// TIA Portal V15.1 export
// export: Created 2024-06-21T08:41:00.046392Z, ExportSetting WithDefaults, DisplayName Totally Integrated Automation Portal, DisplayVersion V15.1 Update 5, DisplayName TIA Portal Openness, DisplayVersion V15.1 Update 5, DisplayName SINAMICS Startdrive Advanced, DisplayVersion V15.1, DisplayName G130, G150, S120, S150, SINAMICS MV, S210, DisplayVersion V15.1, DisplayName G110M, G120, G120C, G120D, G120P, DisplayVersion V15.1, DisplayName STEP 7 Professional, DisplayVersion V15.1 Update 5, DisplayName STEP 7 Safety, DisplayVersion V15.1, DisplayName WinCC Professional, DisplayVersion V15.1 Update 5, DisplayName SIMATIC Visualization Architect, DisplayVersion V15.1
FUNCTION_BLOCK "LPhoneAlarmReqString"   // FB2255, FBD
TITLE = LPhoneAlarmReq
{ S7_Optimized_Access := 'FALSE' }
AUTHOR : VCC
FAMILY : Function
VERSION : 0.1
// =============================================================================
// This Module Handles Phone Alarm Requests
// =============================================================================
// stored: AutoNumber false, IsIECCheckEnabled false, SetENOAutomatically False, UDAEnableTagReadback false
   VAR_INPUT
      I_PhoneAlarmReq1 { ExternalAccessible := 'False'; ExternalVisible := 'False'; ExternalWritable := 'False'} : Bool;   // Request Team Leader Andon From Loading Stn / Request PhoneAlarm For Station / Request PhoneAlarm
      I_PhoneAlarmReq2 { ExternalAccessible := 'False'; ExternalVisible := 'False'; ExternalWritable := 'False'} : Bool;   // Request Maintenance Andon From Loading Stn / Request PhoneAlarm For Station / Request PhoneAlarm
      I_PhoneAlarmReq3 { ExternalAccessible := 'False'; ExternalVisible := 'False'; ExternalWritable := 'False'} : Bool;   // Request PhoneAlarm For Station / Request PhoneAlarm
      I_PhoneAlarmReq4 { ExternalAccessible := 'False'; ExternalVisible := 'False'; ExternalWritable := 'False'} : Bool;   // Request PhoneAlarm For Station / Request PhoneAlarm
      I_PhoneAlarmReq5 { ExternalAccessible := 'False'; ExternalVisible := 'False'; ExternalWritable := 'False'} : Bool;   // Request PhoneAlarm For Station / Request PhoneAlarm
      I_PhoneAlarmReq6 { ExternalAccessible := 'False'; ExternalVisible := 'False'; ExternalWritable := 'False'} : Bool;   // Request PhoneAlarm For Station / Request PhoneAlarm
      I_PhoneAlarmReq7 { ExternalAccessible := 'False'; ExternalVisible := 'False'; ExternalWritable := 'False'} : Bool;   // Request PhoneAlarm For Station / Request PhoneAlarm
      I_PhoneAlarmReq8 { ExternalAccessible := 'False'; ExternalVisible := 'False'; ExternalWritable := 'False'} : Bool;   // Request PhoneAlarm For Station / Request PhoneAlarm
      I_PhoneAlarmReq9 { ExternalAccessible := 'False'; ExternalVisible := 'False'; ExternalWritable := 'False'} : Bool;   // Request PhoneAlarm For Station / Request PhoneAlarm
      I_PhoneAlarmReq10 { ExternalAccessible := 'False'; ExternalVisible := 'False'; ExternalWritable := 'False'} : Bool;   // Request PhoneAlarm For Station / Request PhoneAlarm
      I_PhoneAlarmReq11 { ExternalAccessible := 'False'; ExternalVisible := 'False'; ExternalWritable := 'False'} : Bool;   // Request PhoneAlarm For Station / Request PhoneAlarm
      I_PhoneAlarmReq12 { ExternalAccessible := 'False'; ExternalVisible := 'False'; ExternalWritable := 'False'} : Bool;   // Request PhoneAlarm For Station / Request PhoneAlarm
      I_PhoneAlarmReq13 { ExternalAccessible := 'False'; ExternalVisible := 'False'; ExternalWritable := 'False'} : Bool;   // Request PhoneAlarm For Station / Request PhoneAlarm
      I_PhoneAlarmReq14 { ExternalAccessible := 'False'; ExternalVisible := 'False'; ExternalWritable := 'False'} : Bool;   // Request PhoneAlarm For Station / Request PhoneAlarm
      I_PhoneAlarmReq15 { ExternalAccessible := 'False'; ExternalVisible := 'False'; ExternalWritable := 'False'} : Bool;   // Request PhoneAlarm For Station / Request PhoneAlarm
      I_PhoneAlarmReq16 { ExternalAccessible := 'False'; ExternalVisible := 'False'; ExternalWritable := 'False'} : Bool;   // Request PhoneAlarm For Station / Request PhoneAlarm
      C_MessageType1 { ExternalAccessible := 'False'; ExternalVisible := 'False'; ExternalWritable := 'False'} : String[20];   // Configuration Station / Configuration Message
      C_Message1 { ExternalAccessible := 'False'; ExternalVisible := 'False'; ExternalWritable := 'False'} : String[120];   // Configuration Station / Configuration Message
      C_MessageType2 { ExternalAccessible := 'False'; ExternalVisible := 'False'; ExternalWritable := 'False'} : String[20];   // Configuration Station / Configuration Message
      C_Message2 { ExternalAccessible := 'False'; ExternalVisible := 'False'; ExternalWritable := 'False'} : String[120];   // Configuration Station / Configuration Message
      C_MessageType3 { ExternalAccessible := 'False'; ExternalVisible := 'False'; ExternalWritable := 'False'} : String[20];   // Configuration Station / Configuration Message
      C_Message3 { ExternalAccessible := 'False'; ExternalVisible := 'False'; ExternalWritable := 'False'} : String[120];   // Configuration Station / Configuration Message
      C_MessageType4 { ExternalAccessible := 'False'; ExternalVisible := 'False'; ExternalWritable := 'False'} : String[20];   // Configuration Station / Configuration Message
      C_Message4 { ExternalAccessible := 'False'; ExternalVisible := 'False'; ExternalWritable := 'False'} : String[120];   // Configuration Station / Configuration Message
      C_MessageType5 { ExternalAccessible := 'False'; ExternalVisible := 'False'; ExternalWritable := 'False'} : String[20];   // Configuration Station / Configuration Message
      C_Message5 { ExternalAccessible := 'False'; ExternalVisible := 'False'; ExternalWritable := 'False'} : String[120];   // Configuration Station / Configuration Message
      C_MessageType6 { ExternalAccessible := 'False'; ExternalVisible := 'False'; ExternalWritable := 'False'} : String[20];   // Configuration Station / Configuration Message
      C_Message6 { ExternalAccessible := 'False'; ExternalVisible := 'False'; ExternalWritable := 'False'} : String[120];   // Configuration Station / Configuration Message
      C_MessageType7 { ExternalAccessible := 'False'; ExternalVisible := 'False'; ExternalWritable := 'False'} : String[20];   // Configuration Station / Configuration Message
      C_Message7 { ExternalAccessible := 'False'; ExternalVisible := 'False'; ExternalWritable := 'False'} : String[120];   // Configuration Station / Configuration Message
      C_MessageType8 { ExternalAccessible := 'False'; ExternalVisible := 'False'; ExternalWritable := 'False'} : String[20];   // Configuration Station / Configuration Message
      C_Message8 { ExternalAccessible := 'False'; ExternalVisible := 'False'; ExternalWritable := 'False'} : String[120];   // Configuration Station / Configuration Message
      C_MessageType9 { ExternalAccessible := 'False'; ExternalVisible := 'False'; ExternalWritable := 'False'} : String[20];   // Configuration Station / Configuration Message
      C_Message9 { ExternalAccessible := 'False'; ExternalVisible := 'False'; ExternalWritable := 'False'} : String[120];   // Configuration Station / Configuration Message
      C_MessageType10 { ExternalAccessible := 'False'; ExternalVisible := 'False'; ExternalWritable := 'False'} : String[20];   // Configuration Station / Configuration Message
      C_Message10 { ExternalAccessible := 'False'; ExternalVisible := 'False'; ExternalWritable := 'False'} : String[120];   // Configuration Station / Configuration Message
      C_MessageType11 { ExternalAccessible := 'False'; ExternalVisible := 'False'; ExternalWritable := 'False'} : String[20];   // Configuration Station / Configuration Message
      C_Message11 { ExternalAccessible := 'False'; ExternalVisible := 'False'; ExternalWritable := 'False'} : String[120];   // Configuration Station / Configuration Message
      C_MessageType12 { ExternalAccessible := 'False'; ExternalVisible := 'False'; ExternalWritable := 'False'} : String[20];   // Configuration Station / Configuration Message
      C_Message12 { ExternalAccessible := 'False'; ExternalVisible := 'False'; ExternalWritable := 'False'} : String[120];   // Configuration Station / Configuration Message
      C_MessageType13 { ExternalAccessible := 'False'; ExternalVisible := 'False'; ExternalWritable := 'False'} : String[20];   // Configuration Station / Configuration Message
      C_Message13 { ExternalAccessible := 'False'; ExternalVisible := 'False'; ExternalWritable := 'False'} : String[120];   // Configuration Station / Configuration Message
      C_MessageType14 { ExternalAccessible := 'False'; ExternalVisible := 'False'; ExternalWritable := 'False'} : String[20];   // Configuration Station / Configuration Message
      C_Message14 { ExternalAccessible := 'False'; ExternalVisible := 'False'; ExternalWritable := 'False'} : String[120];   // Configuration Station / Configuration Message
      C_MessageType15 { ExternalAccessible := 'False'; ExternalVisible := 'False'; ExternalWritable := 'False'} : String[20];   // Configuration Station / Configuration Message
      C_Message15 { ExternalAccessible := 'False'; ExternalVisible := 'False'; ExternalWritable := 'False'} : String[120];   // Configuration Station / Configuration Message
      C_MessageType16 { ExternalAccessible := 'False'; ExternalVisible := 'False'; ExternalWritable := 'False'} : String[20];   // Configuration Station / Configuration Message
      C_Message16 { ExternalAccessible := 'False'; ExternalVisible := 'False'; ExternalWritable := 'False'} : String[120];   // Configuration Station / Configuration Message
      C_VDCommRecvDB { ExternalAccessible := 'False'; ExternalVisible := 'False'; ExternalWritable := 'False'} : DB_ANY;   // VD communication system receive DB; Not to be used by application / VD communication system receive DB Not to be used by Application
      C_VDCommSendDB { ExternalAccessible := 'False'; ExternalVisible := 'False'; ExternalWritable := 'False'} : DB_ANY;   // VD communication system send DB; Not to be used by application / VD communication system send DB Not to be used by Application
      C_LocalRecvDB { ExternalAccessible := 'False'; ExternalVisible := 'False'; ExternalWritable := 'False'} : DB_ANY;   // Local DB To Store Received Data
      C_LocalSendDB { ExternalAccessible := 'False'; ExternalVisible := 'False'; ExternalWritable := 'False'} : DB_ANY;   // Local DB for send data; to be used by application / Local DB For Send Data Used By The Application
      C_SubSystem { ExternalAccessible := 'False'; ExternalVisible := 'False'; ExternalWritable := 'False'} : Int;   // Number to identify the subsystem / Identify Subsystem
      C_FilterMessage1 { ExternalAccessible := 'False'; ExternalVisible := 'False'; ExternalWritable := 'False'} : Time;   // Filter
      C_FilterMessage2 { ExternalAccessible := 'False'; ExternalVisible := 'False'; ExternalWritable := 'False'} : Time;   // Filter
      C_FilterMessage3 { ExternalAccessible := 'False'; ExternalVisible := 'False'; ExternalWritable := 'False'} : Time;   // Filter
      C_FilterMessage4 { ExternalAccessible := 'False'; ExternalVisible := 'False'; ExternalWritable := 'False'} : Time;   // Filter
      C_FilterMessage5 { ExternalAccessible := 'False'; ExternalVisible := 'False'; ExternalWritable := 'False'} : Time;   // Filter
      C_FilterMessage6 { ExternalAccessible := 'False'; ExternalVisible := 'False'; ExternalWritable := 'False'} : Time;   // Filter
      C_FilterMessage7 { ExternalAccessible := 'False'; ExternalVisible := 'False'; ExternalWritable := 'False'} : Time;   // Filter
      C_FilterMessage8 { ExternalAccessible := 'False'; ExternalVisible := 'False'; ExternalWritable := 'False'} : Time;   // Filter
      C_FilterMessage9 { ExternalAccessible := 'False'; ExternalVisible := 'False'; ExternalWritable := 'False'} : Time;   // Filter
      C_FilterMessage10 { ExternalAccessible := 'False'; ExternalVisible := 'False'; ExternalWritable := 'False'} : Time;   // Filter
      C_FilterMessage11 { ExternalAccessible := 'False'; ExternalVisible := 'False'; ExternalWritable := 'False'} : Time;   // Filter
      C_FilterMessage12 { ExternalAccessible := 'False'; ExternalVisible := 'False'; ExternalWritable := 'False'} : Time;   // Filter
      C_FilterMessage13 { ExternalAccessible := 'False'; ExternalVisible := 'False'; ExternalWritable := 'False'} : Time;   // Filter
      C_FilterMessage14 { ExternalAccessible := 'False'; ExternalVisible := 'False'; ExternalWritable := 'False'} : Time;   // Filter
      C_FilterMessage15 { ExternalAccessible := 'False'; ExternalVisible := 'False'; ExternalWritable := 'False'} : Time;   // Filter
      C_FilterMessage16 { ExternalAccessible := 'False'; ExternalVisible := 'False'; ExternalWritable := 'False'} : Time;   // Filter
   END_VAR
   VAR_IN_OUT
      IO_VD : "VDComm";   // Communication
      H_HMI : "H_HMI";   // Animation
      H_PhoneAlarmReqString : "H_PhoneAlarmReqString";   // Animation
   END_VAR
   VAR DB_SPECIFIC
      ReqPhoneAlarm { ExternalAccessible := 'False'; ExternalVisible := 'False'; ExternalWritable := 'False'} : Array[1..16] of Bool;   // Request Team Leader Andon / Request PhoneAlarm
      VDReqPhoneAlarm { ExternalAccessible := 'False'; ExternalVisible := 'False'; ExternalWritable := 'False'} : Array[1..16] of Bool;   // VD Request Team Leader Andon / VD Request PhoneAlarm
      Done { ExternalAccessible := 'False'; ExternalVisible := 'False'; ExternalWritable := 'False'} : Array[1..16] of Bool;   // Array
      StnEdge { ExternalAccessible := 'False'; ExternalVisible := 'False'; ExternalWritable := 'False'} : Array[1..16] of Bool;   // Pos Edge
      SendDoneToVD { ExternalAccessible := 'False'; ExternalVisible := 'False'; ExternalWritable := 'False'} : Bool;   // Request Is Finished
      SendVD { ExternalAccessible := 'False'; ExternalVisible := 'False'; ExternalWritable := 'False'} : Bool;   // Send
      PhoneAlarmReqActiveStn1 { ExternalAccessible := 'False'; ExternalVisible := 'False'; ExternalWritable := 'False'} : Bool;   // Indication Request Team Leader Andon / Indication Request
      PhoneAlarmReqActiveStn2 { ExternalAccessible := 'False'; ExternalVisible := 'False'; ExternalWritable := 'False'} : Bool;   // Indication Maintenance Andon / Indication Request
      PhoneAlarmReqActiveStn3 { ExternalAccessible := 'False'; ExternalVisible := 'False'; ExternalWritable := 'False'} : Bool;   // Indication Request
      PhoneAlarmReqActiveStn4 { ExternalAccessible := 'False'; ExternalVisible := 'False'; ExternalWritable := 'False'} : Bool;   // Indication Request
      PhoneAlarmReqActiveStn5 { ExternalAccessible := 'False'; ExternalVisible := 'False'; ExternalWritable := 'False'} : Bool;   // Indication Request
      PhoneAlarmReqActiveStn6 { ExternalAccessible := 'False'; ExternalVisible := 'False'; ExternalWritable := 'False'} : Bool;   // Indication Request
      PhoneAlarmReqActiveStn7 { ExternalAccessible := 'False'; ExternalVisible := 'False'; ExternalWritable := 'False'} : Bool;   // Indication Request
      PhoneAlarmReqActiveStn8 { ExternalAccessible := 'False'; ExternalVisible := 'False'; ExternalWritable := 'False'} : Bool;   // Indication Request
      PhoneAlarmReqActiveStn9 { ExternalAccessible := 'False'; ExternalVisible := 'False'; ExternalWritable := 'False'} : Bool;   // Indication Request
      PhoneAlarmReqActiveStn10 { ExternalAccessible := 'False'; ExternalVisible := 'False'; ExternalWritable := 'False'} : Bool;   // Indication Request
      PhoneAlarmReqActiveStn11 { ExternalAccessible := 'False'; ExternalVisible := 'False'; ExternalWritable := 'False'} : Bool;   // Indication Request
      PhoneAlarmReqActiveStn12 { ExternalAccessible := 'False'; ExternalVisible := 'False'; ExternalWritable := 'False'} : Bool;   // Indication Request
      PhoneAlarmReqActiveStn13 { ExternalAccessible := 'False'; ExternalVisible := 'False'; ExternalWritable := 'False'} : Bool;   // Indication Request
      PhoneAlarmReqActiveStn14 { ExternalAccessible := 'False'; ExternalVisible := 'False'; ExternalWritable := 'False'} : Bool;   // Indication Request
      PhoneAlarmReqActiveStn15 { ExternalAccessible := 'False'; ExternalVisible := 'False'; ExternalWritable := 'False'} : Bool;   // Indication Request
      PhoneAlarmReqActiveStn16 { ExternalAccessible := 'False'; ExternalVisible := 'False'; ExternalWritable := 'False'} : Bool;   // Indication Request
      VDMessage { ExternalAccessible := 'False'; ExternalVisible := 'False'; ExternalWritable := 'False'} : Struct   // VD MEssage to send
         VDMessageType { ExternalAccessible := 'False'; ExternalVisible := 'False'; ExternalWritable := 'False'} : Array[0..19] of Byte;   // Attention Event / VD MessageType
         VDMessage { ExternalAccessible := 'False'; ExternalVisible := 'False'; ExternalWritable := 'False'} : Array[0..119] of Byte;   // Attention Event / VD Message
      END_STRUCT;
   END_VAR
   VAR
      _VDComSubSystem { ExternalAccessible := 'False'; ExternalVisible := 'False'; ExternalWritable := 'False'; S7_SetPoint := 'True'} : "LVDComSubSystemS7-1500";   // FB
   END_VAR
   VAR DB_SPECIFIC
      Edge { ExternalAccessible := 'False'; ExternalVisible := 'False'; ExternalWritable := 'False'} : Array[0..15] of Bool;   // Array Edge
      InitDone { ExternalAccessible := 'False'; ExternalVisible := 'False'; ExternalWritable := 'False'} : Array[1..32] of Bool;   // Init Done
      InitDoneEdge { ExternalAccessible := 'False'; ExternalVisible := 'False'; ExternalWritable := 'False'} : Array[1..32] of Bool;   // Edge Done
      MessageType { ExternalAccessible := 'False'; ExternalVisible := 'False'; ExternalWritable := 'False'} : Int;   // Message Type
      MessageLength { ExternalAccessible := 'False'; ExternalVisible := 'False'; ExternalWritable := 'False'} : Word;   // Message Type / Message Lenght
      _Filter1 { ExternalAccessible := 'False'; ExternalVisible := 'False'; ExternalWritable := 'False'; S7_SetPoint := 'True'} : TON_TIME;   // FB
      _Filter2 { ExternalAccessible := 'False'; ExternalVisible := 'False'; ExternalWritable := 'False'; S7_SetPoint := 'True'} : TON_TIME;   // FB
      _Filter3 { ExternalAccessible := 'False'; ExternalVisible := 'False'; ExternalWritable := 'False'; S7_SetPoint := 'True'} : TON_TIME;   // FB
      _Filter4 { ExternalAccessible := 'False'; ExternalVisible := 'False'; ExternalWritable := 'False'; S7_SetPoint := 'True'} : TON_TIME;   // FB
      _Filter5 { ExternalAccessible := 'False'; ExternalVisible := 'False'; ExternalWritable := 'False'; S7_SetPoint := 'True'} : TON_TIME;   // FB
      _Filter6 { ExternalAccessible := 'False'; ExternalVisible := 'False'; ExternalWritable := 'False'; S7_SetPoint := 'True'} : TON_TIME;   // FB
      _Filter7 { ExternalAccessible := 'False'; ExternalVisible := 'False'; ExternalWritable := 'False'; S7_SetPoint := 'True'} : TON_TIME;   // FB
      _Filter8 { ExternalAccessible := 'False'; ExternalVisible := 'False'; ExternalWritable := 'False'; S7_SetPoint := 'True'} : TON_TIME;   // FB
      _Filter9 { ExternalAccessible := 'False'; ExternalVisible := 'False'; ExternalWritable := 'False'; S7_SetPoint := 'True'} : TON_TIME;   // FB
      _Filter10 { ExternalAccessible := 'False'; ExternalVisible := 'False'; ExternalWritable := 'False'; S7_SetPoint := 'True'} : TON_TIME;   // FB
      _Filter11 { ExternalAccessible := 'False'; ExternalVisible := 'False'; ExternalWritable := 'False'; S7_SetPoint := 'True'} : TON_TIME;   // FB
      _Filter12 { ExternalAccessible := 'False'; ExternalVisible := 'False'; ExternalWritable := 'False'; S7_SetPoint := 'True'} : TON_TIME;   // FB
      _Filter13 { ExternalAccessible := 'False'; ExternalVisible := 'False'; ExternalWritable := 'False'; S7_SetPoint := 'True'} : TON_TIME;   // FB
      _Filter14 { ExternalAccessible := 'False'; ExternalVisible := 'False'; ExternalWritable := 'False'; S7_SetPoint := 'True'} : TON_TIME;   // FB
      _Filter15 { ExternalAccessible := 'False'; ExternalVisible := 'False'; ExternalWritable := 'False'; S7_SetPoint := 'True'} : TON_TIME;   // FB
      _Filter16 { ExternalAccessible := 'False'; ExternalVisible := 'False'; ExternalWritable := 'False'; S7_SetPoint := 'True'} : TON_TIME;   // FB
      SendToVDTimeOut { ExternalAccessible := 'False'; ExternalVisible := 'False'; ExternalWritable := 'False'; S7_SetPoint := 'True'} : TON_TIME;   // Send to VD time-out
      ResetVDComm { ExternalAccessible := 'False'; ExternalVisible := 'False'; ExternalWritable := 'False'} : Bool;   // Reset VD communication upon timeout
      VDMessageTypeTemp { ExternalAccessible := 'False'; ExternalVisible := 'False'; ExternalWritable := 'False'} : String[20];   // Attention Event / VDMessageTypeTemp string 20 characters
      VDMessageTemp { ExternalAccessible := 'False'; ExternalVisible := 'False'; ExternalWritable := 'False'} : String[120];   // Attention Event / VDMessageTemp string 120 characters
      VDMessageTypeSerialzePos { ExternalAccessible := 'False'; ExternalVisible := 'False'; ExternalWritable := 'False'} : DInt;   // Serialize position
      VDMessageSerialzePos { ExternalAccessible := 'False'; ExternalVisible := 'False'; ExternalWritable := 'False'} : DInt;   // Serialize position
      VDMessageTypeTempArray { ExternalAccessible := 'False'; ExternalVisible := 'False'; ExternalWritable := 'False'} : Array[0..21] of Byte;   // VDMessageType Array
      VDMessageTempArray { ExternalAccessible := 'False'; ExternalVisible := 'False'; ExternalWritable := 'False'} : Array[0..121] of Byte;   // VDMessage Array
   END_VAR
   VAR_TEMP
      RequestCommand1 : Bool;   // Light On To Building Infrastructure / Request Configured Command
      RequestCommand2 : Bool;   // Light On To Building Infrastructure / Request Configured Command
      RequestCommand3 : Bool;   // Light On To Building Infrastructure / Request Configured Command
      RequestCommand4 : Bool;   // Light On To Building Infrastructure / Request Configured Command
      RequestCommand5 : Bool;   // Light On To Building Infrastructure / Request Configured Command
      RequestCommand6 : Bool;   // Light On To Building Infrastructure / Request Configured Command
      RequestCommand7 : Bool;   // Light On To Building Infrastructure / Request Configured Command
      RequestCommand8 : Bool;   // Light On To Building Infrastructure / Request Configured Command
      RequestCommand9 : Bool;   // Request Configured Command
      RequestCommand10 : Bool;   // Request Configured Command
      RequestCommand11 : Bool;   // Request Configured Command
      RequestCommand12 : Bool;   // Request Configured Command
      RequestCommand13 : Bool;   // Request Configured Command
      RequestCommand14 : Bool;   // Request Configured Command
      RequestCommand15 : Bool;   // Request Configured Command
      RequestCommand16 : Bool;   // Request Configured Command
      RecvDBNbr : Int;   // Receive system DB Number
      SendDBNbr : Int;   // Send system DB Number
      LocalRecvDBNbr : Int;   // Receive DB Number Local by Application
      LocalSendDBNbr : Int;   // Send DB Number Local by Application
      PtrASnd : Any;   // Pointer to the Application receive DB / Pointer to the Application send DB
   END_VAR
   VAR CONSTANT
      String20Spaces : String := '                    ';   // String with 20 spaces
      String120Spaces : String := '                                                                                                                        ';   // String with 120 spaces
   END_VAR
   VAR_TEMP   // added for the SCL form of the ladder/FBD networks
      _w1 : Bool;
      _w2 : Bool;
   END_VAR
BEGIN

REGION Network 1: **** 1 - Inputs **** Extract The Commands From HMI
   // Extract The Commands From HMI
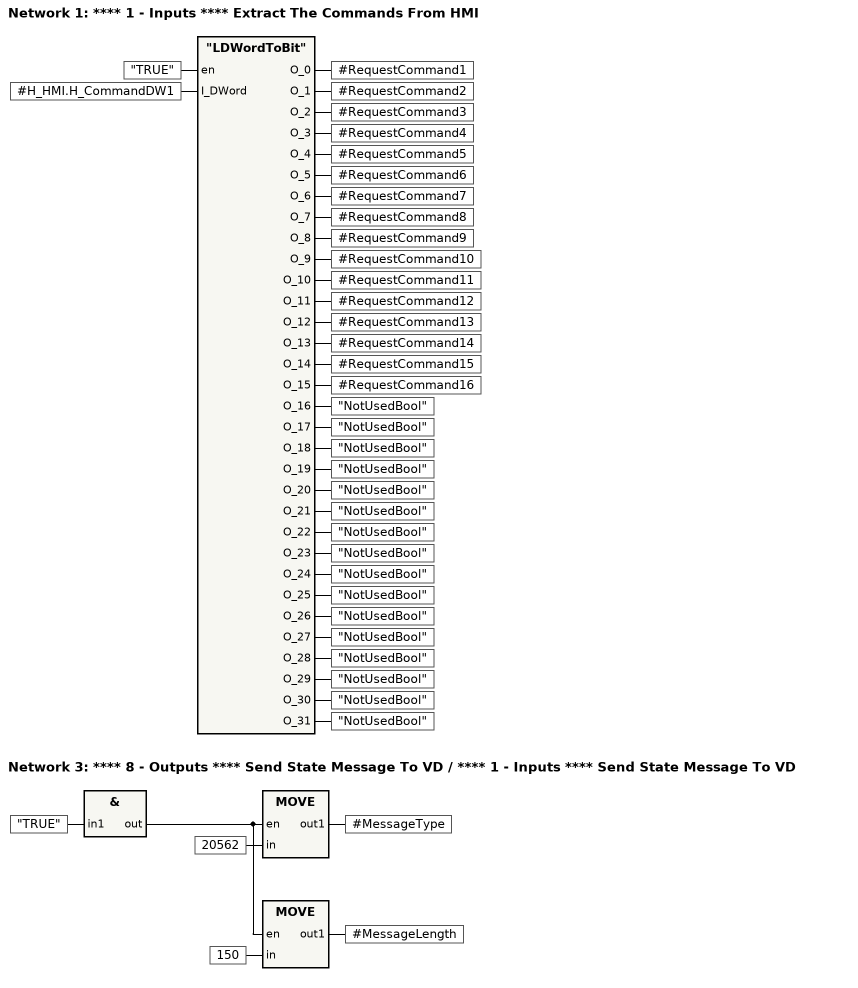
   IF "TRUE" THEN
       "LDWordToBit"(I_DWord := #H_HMI.H_CommandDW1,
                     O_0 => #RequestCommand1,
                     O_1 => #RequestCommand2,
                     O_2 => #RequestCommand3,
                     O_3 => #RequestCommand4,
                     O_4 => #RequestCommand5,
                     O_5 => #RequestCommand6,
                     O_6 => #RequestCommand7,
                     O_7 => #RequestCommand8,
                     O_8 => #RequestCommand9,
                     O_9 => #RequestCommand10,
                     O_10 => #RequestCommand11,
                     O_11 => #RequestCommand12,
                     O_12 => #RequestCommand13,
                     O_13 => #RequestCommand14,
                     O_14 => #RequestCommand15,
                     O_15 => #RequestCommand16,
                     O_16 => "NotUsedBool",
                     O_17 => "NotUsedBool",
                     O_18 => "NotUsedBool",
                     O_19 => "NotUsedBool",
                     O_20 => "NotUsedBool",
                     O_21 => "NotUsedBool",
                     O_22 => "NotUsedBool",
                     O_23 => "NotUsedBool",
                     O_24 => "NotUsedBool",
                     O_25 => "NotUsedBool",
                     O_26 => "NotUsedBool",
                     O_27 => "NotUsedBool",
                     O_28 => "NotUsedBool",
                     O_29 => "NotUsedBool",
                     O_30 => "NotUsedBool",
                     O_31 => "NotUsedBool");
   END_IF;
END_REGION

NETWORK
TITLE = **** 1 - Inputs **** Load DB / **** 1 - Inputs **** Load DB number
// Load DB numbers to local variables from the Receive and Send DB from - VD Master - VD Subsystem
// Read DB Number Recv
      OPN   #C_VDCommRecvDB;
      L     DBNO;
      T     #RecvDBNbr;

// Read DB Number Send
      OPN   #C_VDCommSendDB;
      L     DBNO;
      T     #SendDBNbr;

// DB Number from VD Sub system
      OPN   #C_LocalRecvDB;
      L     DBNO;
      T     #LocalRecvDBNbr;

// Read DB Number Send
      OPN   #C_LocalSendDB;
      L     DBNO;
      T     #LocalSendDBNbr;

REGION Network 3: **** 8 - Outputs **** Send State Message To VD / **** 1 - Inputs **** Send State Message To VD
   // Send State Message To VD
   IF "TRUE" THEN
       #MessageType := 20562;
       #MessageLength := 150;
   END_IF;
END_REGION

REGION Network 4: **** 3.1 - Communication - Other Systems **** Send Message
   // Send Message
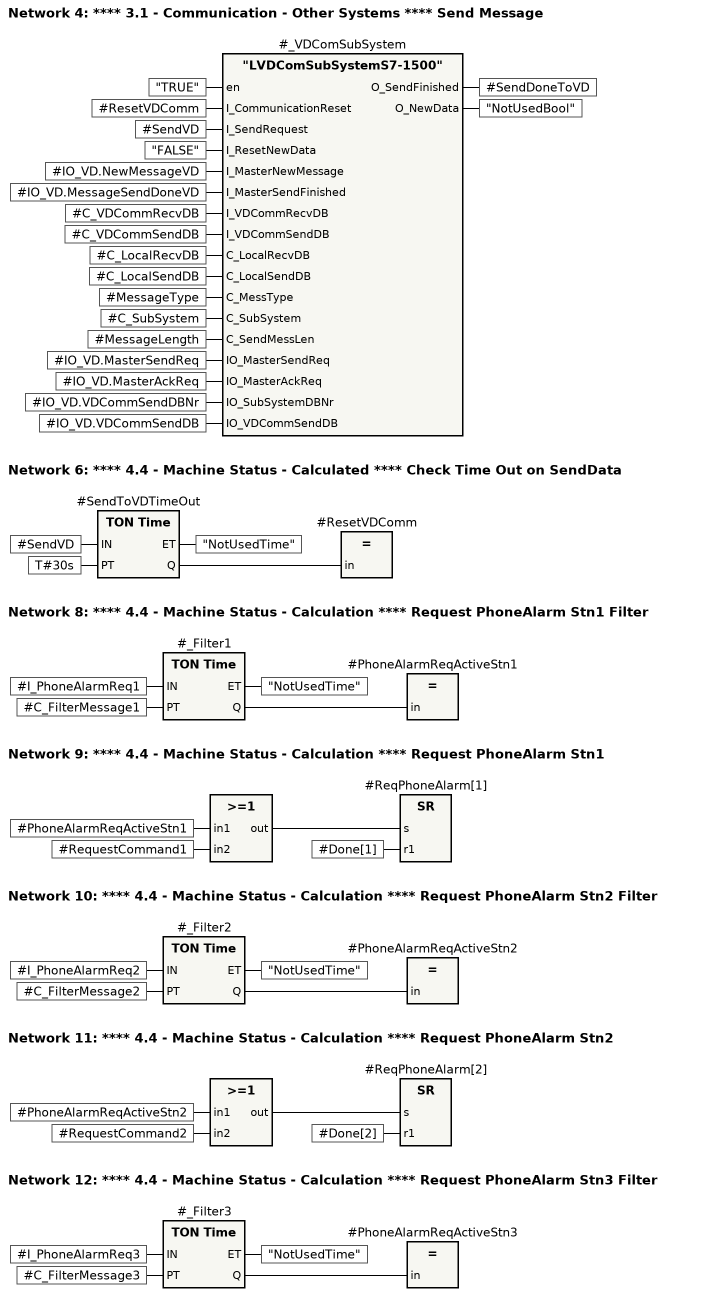
   IF "TRUE" THEN
       #_VDComSubSystem(I_CommunicationReset := #ResetVDComm,   // "LVDComSubSystemS7-1500"
                        I_SendRequest := #SendVD,
                        I_ResetNewData := "FALSE",
                        I_MasterNewMessage := #IO_VD.NewMessageVD,
                        I_MasterSendFinished := #IO_VD.MessageSendDoneVD,
                        I_VDCommRecvDB := #C_VDCommRecvDB,
                        I_VDCommSendDB := #C_VDCommSendDB,
                        C_LocalRecvDB := #C_LocalRecvDB,
                        C_LocalSendDB := #C_LocalSendDB,
                        C_MessType := #MessageType,
                        C_SubSystem := #C_SubSystem,
                        C_SendMessLen := #MessageLength,
                        IO_MasterSendReq := #IO_VD.MasterSendReq,
                        IO_MasterAckReq := #IO_VD.MasterAckReq,
                        IO_SubSystemDBNr := #IO_VD.VDCommSendDBNr,
                        IO_VDCommSendDB := #IO_VD.VDCommSendDB,
                        O_SendFinished => #SendDoneToVD,
                        O_NewData => "NotUsedBool");
   END_IF;
END_REGION

NETWORK
TITLE = **** 3.1 - Communication - Other Systems **** Configure DB / **** 4.2 Parameter **** Configure DB
// Configure DB pointers
      LAR1  P##PtrASnd;
      L     16#1002;  // Data type to copy B#16#2 = Bytes
      T     LW [AR1, P#0.0];
      L     #MessageLength;  //Length sending data
      T     LW [AR1, P#2.0];
      L     #LocalSendDBNbr;  // Local Send DB Number
      T     LW [AR1, P#4.0];
      L     10;  // Offset in DB (skip VD header)
      SLD   3;  // Convert to pointer - Shift Left DW
      OD    16#8400_0000;  // Memory area DB Memory - 84 equals DB
      T     LD [AR1, P#6.0];


REGION Network 6: **** 4.4 - Machine Status - Calculated **** Check Time Out on SendData
   // Reset Send request when time out elapses
   // Reset the VD communication
   #SendToVDTimeOut(IN := #SendVD, PT := T#30s, ET => "NotUsedTime");   // TON
   #ResetVDComm := #SendToVDTimeOut.Q;
END_REGION

NETWORK
TITLE = **** 4.4 - Machine status - Calculated **** Init Done
// Init Done

      A     #I_PhoneAlarmReq1;
      O     #RequestCommand1;
      FP    #InitDoneEdge[1];
      =     #InitDone[1];

      A     #I_PhoneAlarmReq2;
      O     #RequestCommand2;
      FP    #InitDoneEdge[2];
      =     #InitDone[2];

      A     #I_PhoneAlarmReq3;
      O     #RequestCommand3;
      FP    #InitDoneEdge[3];
      =     #InitDone[3];

      A     #I_PhoneAlarmReq4;
      O     #RequestCommand4;
      FP    #InitDoneEdge[4];
      =     #InitDone[4];

      A     #I_PhoneAlarmReq5;
      O     #RequestCommand5;
      FP    #InitDoneEdge[5];
      =     #InitDone[5];

      A     #I_PhoneAlarmReq6;
      O     #RequestCommand6;
      FP    #InitDoneEdge[6];
      =     #InitDone[6];

      A     #I_PhoneAlarmReq7;
      O     #RequestCommand7;
      FP    #InitDoneEdge[7];
      =     #InitDone[7];

      A     #I_PhoneAlarmReq8;
      O     #RequestCommand8;
      FP    #InitDoneEdge[8];
      =     #InitDone[8];

      A     #I_PhoneAlarmReq9;
      O     #RequestCommand9;
      FP    #InitDoneEdge[9];
      =     #InitDone[9];

      A     #I_PhoneAlarmReq10;
      O     #RequestCommand10;
      FP    #InitDoneEdge[10];
      =     #InitDone[10];

      A     #I_PhoneAlarmReq11;
      O     #RequestCommand11;
      FP    #InitDoneEdge[11];
      =     #InitDone[11];

      A     #I_PhoneAlarmReq12;
      O     #RequestCommand12;
      FP    #InitDoneEdge[12];
      =     #InitDone[12];

      A     #I_PhoneAlarmReq13;
      O     #RequestCommand13;
      FP    #InitDoneEdge[13];
      =     #InitDone[13];

      A     #I_PhoneAlarmReq14;
      O     #RequestCommand14;
      FP    #InitDoneEdge[14];
      =     #InitDone[14];

      A     #I_PhoneAlarmReq15;
      O     #RequestCommand15;
      FP    #InitDoneEdge[15];
      =     #InitDone[15];

      A     #I_PhoneAlarmReq16;
      O     #RequestCommand16;
      FP    #InitDoneEdge[16];
      =     #InitDone[16];


REGION Network 8: **** 4.4 - Machine Status - Calculation **** Request PhoneAlarm Stn1 Filter
   // Filter
   #_Filter1(IN := #I_PhoneAlarmReq1, PT := #C_FilterMessage1, ET => "NotUsedTime");   // TON
   #PhoneAlarmReqActiveStn1 := #_Filter1.Q;
END_REGION

REGION Network 9: **** 4.4 - Machine Status - Calculation **** Request PhoneAlarm Stn1
   // Request PhoneAlarm Stn1
   IF #PhoneAlarmReqActiveStn1 OR #RequestCommand1 THEN
       #ReqPhoneAlarm[1] := TRUE;   // SR flip-flop
   END_IF;
   IF #Done[1] THEN #ReqPhoneAlarm[1] := FALSE; END_IF;
END_REGION

REGION Network 10: **** 4.4 - Machine Status - Calculation **** Request PhoneAlarm Stn2 Filter
   // Filter
   #_Filter2(IN := #I_PhoneAlarmReq2, PT := #C_FilterMessage2, ET => "NotUsedTime");   // TON
   #PhoneAlarmReqActiveStn2 := #_Filter2.Q;
END_REGION

REGION Network 11: **** 4.4 - Machine Status - Calculation **** Request PhoneAlarm Stn2
   // Request PhoneAlarm Stn2
   IF #PhoneAlarmReqActiveStn2 OR #RequestCommand2 THEN
       #ReqPhoneAlarm[2] := TRUE;   // SR flip-flop
   END_IF;
   IF #Done[2] THEN #ReqPhoneAlarm[2] := FALSE; END_IF;
END_REGION

REGION Network 12: **** 4.4 - Machine Status - Calculation **** Request PhoneAlarm Stn3 Filter
   // Filter
   #_Filter3(IN := #I_PhoneAlarmReq3, PT := #C_FilterMessage3, ET => "NotUsedTime");   // TON
   #PhoneAlarmReqActiveStn3 := #_Filter3.Q;
END_REGION

REGION Network 13: **** 4.4 - Machine Status - Calculation **** Request PhoneAlarm Stn3
   // Request PhoneAlarm Stn3
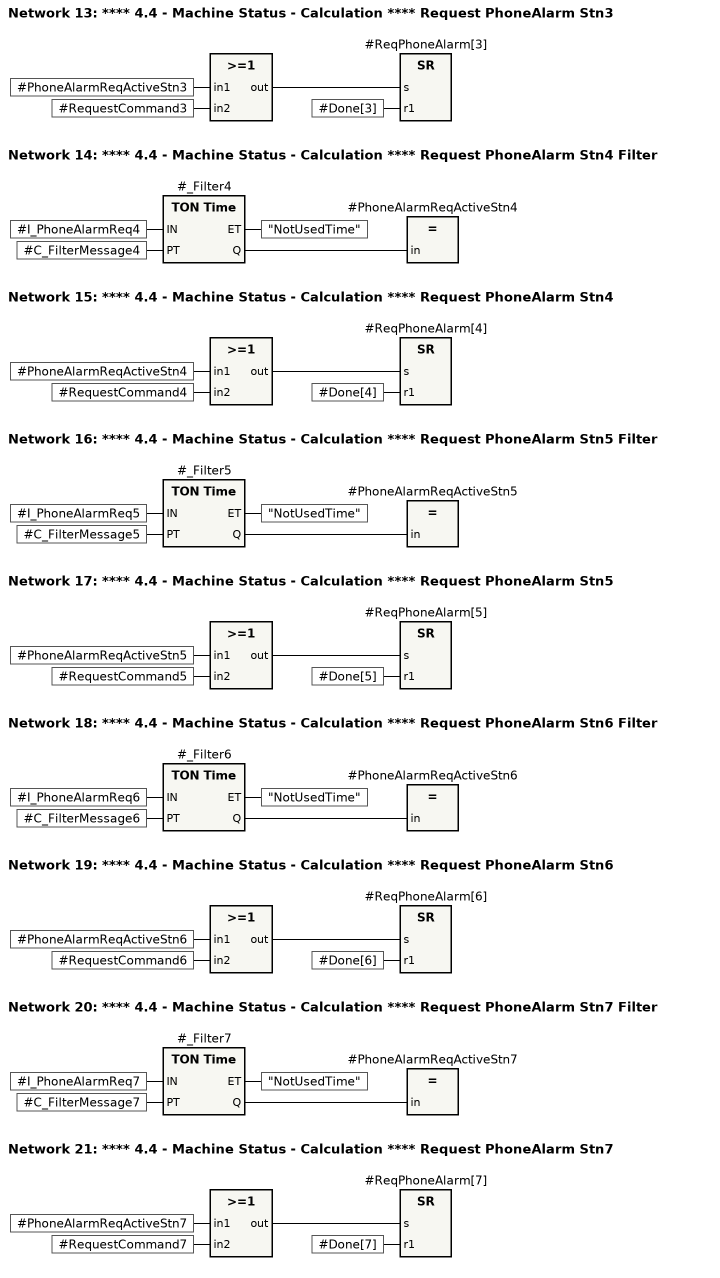
   IF #PhoneAlarmReqActiveStn3 OR #RequestCommand3 THEN
       #ReqPhoneAlarm[3] := TRUE;   // SR flip-flop
   END_IF;
   IF #Done[3] THEN #ReqPhoneAlarm[3] := FALSE; END_IF;
END_REGION

REGION Network 14: **** 4.4 - Machine Status - Calculation **** Request PhoneAlarm Stn4 Filter
   // Filter
   #_Filter4(IN := #I_PhoneAlarmReq4, PT := #C_FilterMessage4, ET => "NotUsedTime");   // TON
   #PhoneAlarmReqActiveStn4 := #_Filter4.Q;
END_REGION

REGION Network 15: **** 4.4 - Machine Status - Calculation **** Request PhoneAlarm Stn4
   // Request PhoneAlarm Stn4
   IF #PhoneAlarmReqActiveStn4 OR #RequestCommand4 THEN
       #ReqPhoneAlarm[4] := TRUE;   // SR flip-flop
   END_IF;
   IF #Done[4] THEN #ReqPhoneAlarm[4] := FALSE; END_IF;
END_REGION

REGION Network 16: **** 4.4 - Machine Status - Calculation **** Request PhoneAlarm Stn5 Filter
   // Filter
   #_Filter5(IN := #I_PhoneAlarmReq5, PT := #C_FilterMessage5, ET => "NotUsedTime");   // TON
   #PhoneAlarmReqActiveStn5 := #_Filter5.Q;
END_REGION

REGION Network 17: **** 4.4 - Machine Status - Calculation **** Request PhoneAlarm Stn5
   // Request PhoneAlarm Stn5
   IF #PhoneAlarmReqActiveStn5 OR #RequestCommand5 THEN
       #ReqPhoneAlarm[5] := TRUE;   // SR flip-flop
   END_IF;
   IF #Done[5] THEN #ReqPhoneAlarm[5] := FALSE; END_IF;
END_REGION

REGION Network 18: **** 4.4 - Machine Status - Calculation **** Request PhoneAlarm Stn6 Filter
   // Filter
   #_Filter6(IN := #I_PhoneAlarmReq6, PT := #C_FilterMessage6, ET => "NotUsedTime");   // TON
   #PhoneAlarmReqActiveStn6 := #_Filter6.Q;
END_REGION

REGION Network 19: **** 4.4 - Machine Status - Calculation **** Request PhoneAlarm Stn6
   // Request PhoneAlarm Stn6
   IF #PhoneAlarmReqActiveStn6 OR #RequestCommand6 THEN
       #ReqPhoneAlarm[6] := TRUE;   // SR flip-flop
   END_IF;
   IF #Done[6] THEN #ReqPhoneAlarm[6] := FALSE; END_IF;
END_REGION

REGION Network 20: **** 4.4 - Machine Status - Calculation **** Request PhoneAlarm Stn7 Filter
   // Filter
   #_Filter7(IN := #I_PhoneAlarmReq7, PT := #C_FilterMessage7, ET => "NotUsedTime");   // TON
   #PhoneAlarmReqActiveStn7 := #_Filter7.Q;
END_REGION

REGION Network 21: **** 4.4 - Machine Status - Calculation **** Request PhoneAlarm Stn7
   // Request PhoneAlarm Stn7
   IF #PhoneAlarmReqActiveStn7 OR #RequestCommand7 THEN
       #ReqPhoneAlarm[7] := TRUE;   // SR flip-flop
   END_IF;
   IF #Done[7] THEN #ReqPhoneAlarm[7] := FALSE; END_IF;
END_REGION

REGION Network 22: **** 4.4 - Machine Status - Calculation **** Request PhoneAlarm Stn8 Filter
   // Filter
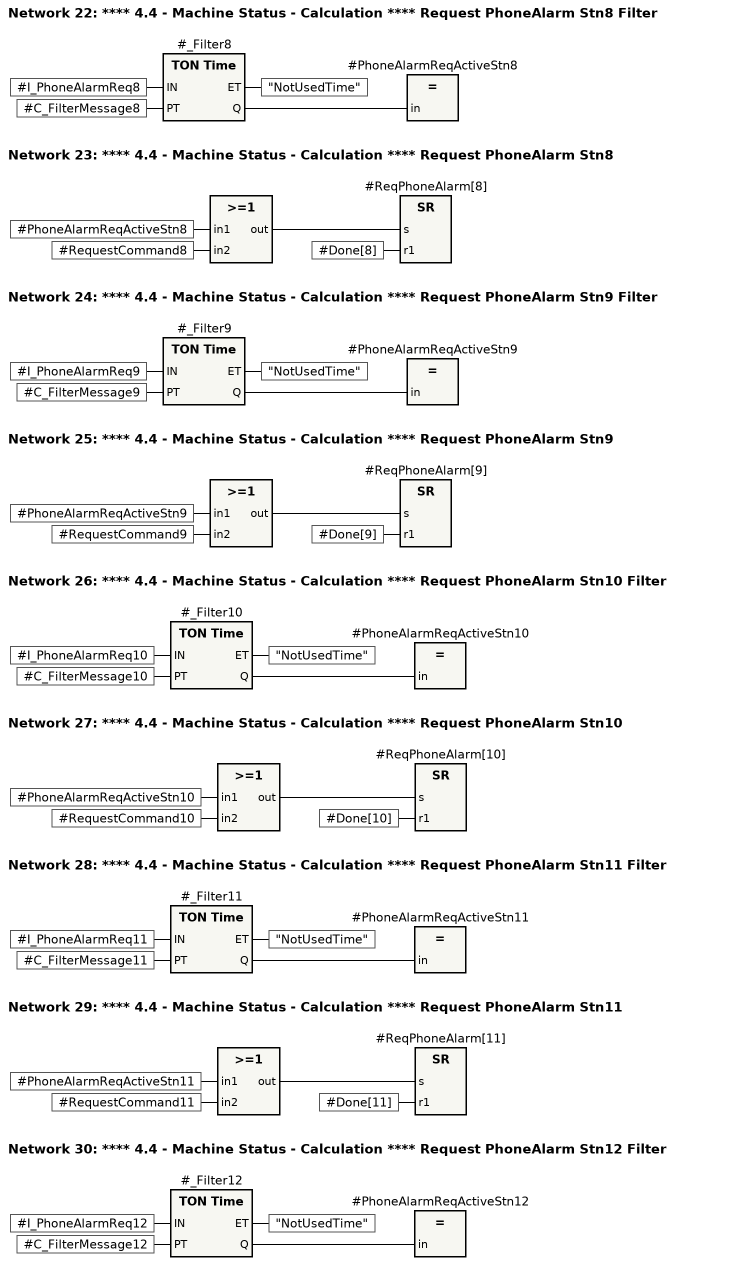
   #_Filter8(IN := #I_PhoneAlarmReq8, PT := #C_FilterMessage8, ET => "NotUsedTime");   // TON
   #PhoneAlarmReqActiveStn8 := #_Filter8.Q;
END_REGION

REGION Network 23: **** 4.4 - Machine Status - Calculation **** Request PhoneAlarm Stn8
   // Request PhoneAlarm Stn8
   IF #PhoneAlarmReqActiveStn8 OR #RequestCommand8 THEN
       #ReqPhoneAlarm[8] := TRUE;   // SR flip-flop
   END_IF;
   IF #Done[8] THEN #ReqPhoneAlarm[8] := FALSE; END_IF;
END_REGION

REGION Network 24: **** 4.4 - Machine Status - Calculation **** Request PhoneAlarm Stn9 Filter
   // Filter
   #_Filter9(IN := #I_PhoneAlarmReq9, PT := #C_FilterMessage9, ET => "NotUsedTime");   // TON
   #PhoneAlarmReqActiveStn9 := #_Filter9.Q;
END_REGION

REGION Network 25: **** 4.4 - Machine Status - Calculation **** Request PhoneAlarm Stn9
   // Request PhoneAlarm Stn9
   IF #PhoneAlarmReqActiveStn9 OR #RequestCommand9 THEN
       #ReqPhoneAlarm[9] := TRUE;   // SR flip-flop
   END_IF;
   IF #Done[9] THEN #ReqPhoneAlarm[9] := FALSE; END_IF;
END_REGION

REGION Network 26: **** 4.4 - Machine Status - Calculation **** Request PhoneAlarm Stn10 Filter
   // Filter
   #_Filter10(IN := #I_PhoneAlarmReq10, PT := #C_FilterMessage10, ET => "NotUsedTime");   // TON
   #PhoneAlarmReqActiveStn10 := #_Filter10.Q;
END_REGION

REGION Network 27: **** 4.4 - Machine Status - Calculation **** Request PhoneAlarm Stn10
   // Request PhoneAlarm Stn10
   IF #PhoneAlarmReqActiveStn10 OR #RequestCommand10 THEN
       #ReqPhoneAlarm[10] := TRUE;   // SR flip-flop
   END_IF;
   IF #Done[10] THEN #ReqPhoneAlarm[10] := FALSE; END_IF;
END_REGION

REGION Network 28: **** 4.4 - Machine Status - Calculation **** Request PhoneAlarm Stn11 Filter
   // Filter
   #_Filter11(IN := #I_PhoneAlarmReq11, PT := #C_FilterMessage11, ET => "NotUsedTime");   // TON
   #PhoneAlarmReqActiveStn11 := #_Filter11.Q;
END_REGION

REGION Network 29: **** 4.4 - Machine Status - Calculation **** Request PhoneAlarm Stn11
   // Request PhoneAlarm Stn11
   IF #PhoneAlarmReqActiveStn11 OR #RequestCommand11 THEN
       #ReqPhoneAlarm[11] := TRUE;   // SR flip-flop
   END_IF;
   IF #Done[11] THEN #ReqPhoneAlarm[11] := FALSE; END_IF;
END_REGION

REGION Network 30: **** 4.4 - Machine Status - Calculation **** Request PhoneAlarm Stn12 Filter
   // Filter
   #_Filter12(IN := #I_PhoneAlarmReq12, PT := #C_FilterMessage12, ET => "NotUsedTime");   // TON
   #PhoneAlarmReqActiveStn12 := #_Filter12.Q;
END_REGION

REGION Network 31: **** 4.4 - Machine Status - Calculation **** Request PhoneAlarm Stn12
   // Request PhoneAlarm Stn12
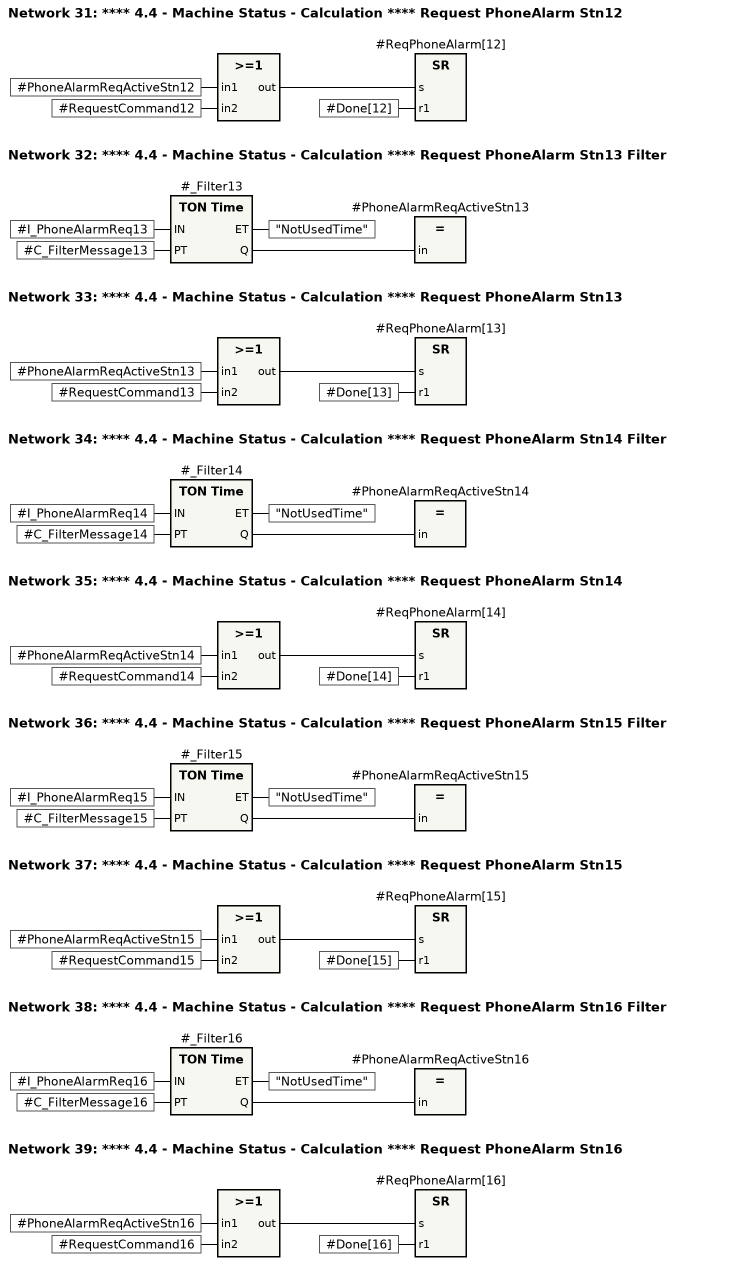
   IF #PhoneAlarmReqActiveStn12 OR #RequestCommand12 THEN
       #ReqPhoneAlarm[12] := TRUE;   // SR flip-flop
   END_IF;
   IF #Done[12] THEN #ReqPhoneAlarm[12] := FALSE; END_IF;
END_REGION

REGION Network 32: **** 4.4 - Machine Status - Calculation **** Request PhoneAlarm Stn13 Filter
   // Filter
   #_Filter13(IN := #I_PhoneAlarmReq13, PT := #C_FilterMessage13, ET => "NotUsedTime");   // TON
   #PhoneAlarmReqActiveStn13 := #_Filter13.Q;
END_REGION

REGION Network 33: **** 4.4 - Machine Status - Calculation **** Request PhoneAlarm Stn13
   // Request PhoneAlarm Stn13
   IF #PhoneAlarmReqActiveStn13 OR #RequestCommand13 THEN
       #ReqPhoneAlarm[13] := TRUE;   // SR flip-flop
   END_IF;
   IF #Done[13] THEN #ReqPhoneAlarm[13] := FALSE; END_IF;
END_REGION

REGION Network 34: **** 4.4 - Machine Status - Calculation **** Request PhoneAlarm Stn14 Filter
   // Filter
   #_Filter14(IN := #I_PhoneAlarmReq14, PT := #C_FilterMessage14, ET => "NotUsedTime");   // TON
   #PhoneAlarmReqActiveStn14 := #_Filter14.Q;
END_REGION

REGION Network 35: **** 4.4 - Machine Status - Calculation **** Request PhoneAlarm Stn14
   // Request PhoneAlarm Stn14
   IF #PhoneAlarmReqActiveStn14 OR #RequestCommand14 THEN
       #ReqPhoneAlarm[14] := TRUE;   // SR flip-flop
   END_IF;
   IF #Done[14] THEN #ReqPhoneAlarm[14] := FALSE; END_IF;
END_REGION

REGION Network 36: **** 4.4 - Machine Status - Calculation **** Request PhoneAlarm Stn15 Filter
   // Filter
   #_Filter15(IN := #I_PhoneAlarmReq15, PT := #C_FilterMessage15, ET => "NotUsedTime");   // TON
   #PhoneAlarmReqActiveStn15 := #_Filter15.Q;
END_REGION

REGION Network 37: **** 4.4 - Machine Status - Calculation **** Request PhoneAlarm Stn15
   // Request PhoneAlarm Stn15
   IF #PhoneAlarmReqActiveStn15 OR #RequestCommand15 THEN
       #ReqPhoneAlarm[15] := TRUE;   // SR flip-flop
   END_IF;
   IF #Done[15] THEN #ReqPhoneAlarm[15] := FALSE; END_IF;
END_REGION

REGION Network 38: **** 4.4 - Machine Status - Calculation **** Request PhoneAlarm Stn16 Filter
   // Filter
   #_Filter16(IN := #I_PhoneAlarmReq16, PT := #C_FilterMessage16, ET => "NotUsedTime");   // TON
   #PhoneAlarmReqActiveStn16 := #_Filter16.Q;
END_REGION

REGION Network 39: **** 4.4 - Machine Status - Calculation **** Request PhoneAlarm Stn16
   // Request PhoneAlarm Stn16
   IF #PhoneAlarmReqActiveStn16 OR #RequestCommand16 THEN
       #ReqPhoneAlarm[16] := TRUE;   // SR flip-flop
   END_IF;
   IF #Done[16] THEN #ReqPhoneAlarm[16] := FALSE; END_IF;
END_REGION

REGION Network 40: **** 4.4 - Machine Status - Calculation **** Message Request Done
   // Message Request Done
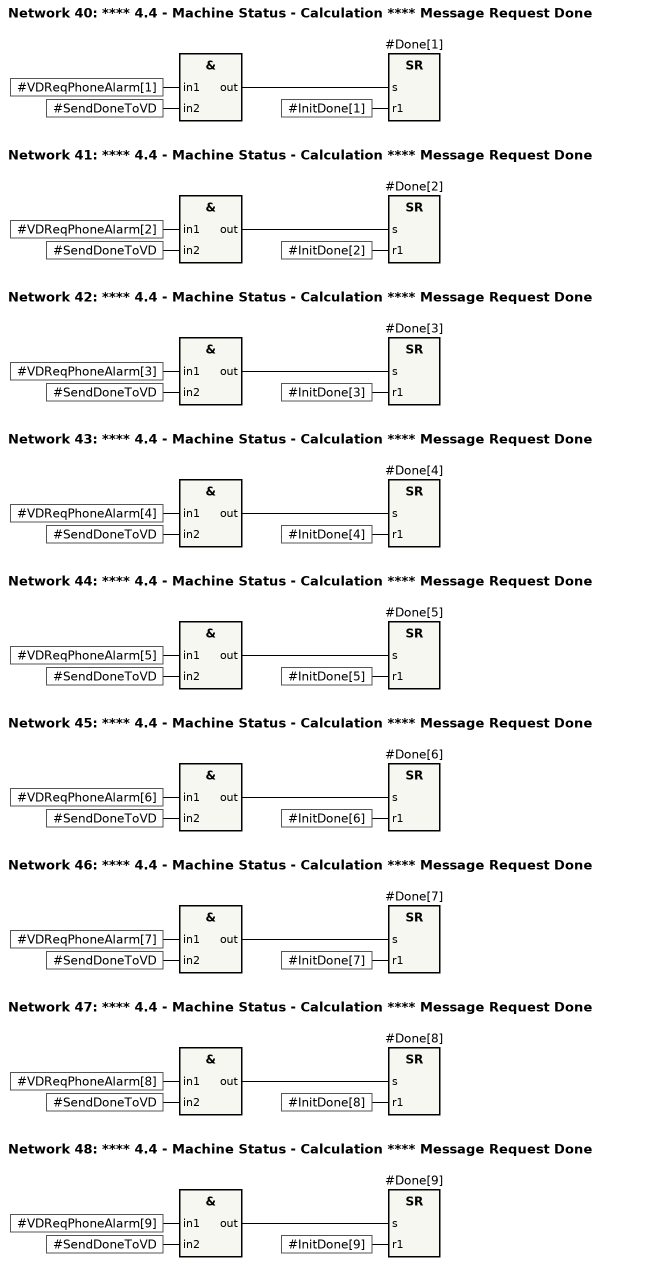
   IF #VDReqPhoneAlarm[1] AND #SendDoneToVD THEN
       #Done[1] := TRUE;   // SR flip-flop
   END_IF;
   IF #InitDone[1] THEN #Done[1] := FALSE; END_IF;
END_REGION

REGION Network 41: **** 4.4 - Machine Status - Calculation **** Message Request Done
   // Message Request Done
   IF #VDReqPhoneAlarm[2] AND #SendDoneToVD THEN
       #Done[2] := TRUE;   // SR flip-flop
   END_IF;
   IF #InitDone[2] THEN #Done[2] := FALSE; END_IF;
END_REGION

REGION Network 42: **** 4.4 - Machine Status - Calculation **** Message Request Done
   // Message Request Done
   IF #VDReqPhoneAlarm[3] AND #SendDoneToVD THEN
       #Done[3] := TRUE;   // SR flip-flop
   END_IF;
   IF #InitDone[3] THEN #Done[3] := FALSE; END_IF;
END_REGION

REGION Network 43: **** 4.4 - Machine Status - Calculation **** Message Request Done
   // Message Request Done
   IF #VDReqPhoneAlarm[4] AND #SendDoneToVD THEN
       #Done[4] := TRUE;   // SR flip-flop
   END_IF;
   IF #InitDone[4] THEN #Done[4] := FALSE; END_IF;
END_REGION

REGION Network 44: **** 4.4 - Machine Status - Calculation **** Message Request Done
   // Message Request Done
   IF #VDReqPhoneAlarm[5] AND #SendDoneToVD THEN
       #Done[5] := TRUE;   // SR flip-flop
   END_IF;
   IF #InitDone[5] THEN #Done[5] := FALSE; END_IF;
END_REGION

REGION Network 45: **** 4.4 - Machine Status - Calculation **** Message Request Done
   // Message Request Done
   IF #VDReqPhoneAlarm[6] AND #SendDoneToVD THEN
       #Done[6] := TRUE;   // SR flip-flop
   END_IF;
   IF #InitDone[6] THEN #Done[6] := FALSE; END_IF;
END_REGION

REGION Network 46: **** 4.4 - Machine Status - Calculation **** Message Request Done
   // Message Request Done
   IF #VDReqPhoneAlarm[7] AND #SendDoneToVD THEN
       #Done[7] := TRUE;   // SR flip-flop
   END_IF;
   IF #InitDone[7] THEN #Done[7] := FALSE; END_IF;
END_REGION

REGION Network 47: **** 4.4 - Machine Status - Calculation **** Message Request Done
   // Message Request Done
   IF #VDReqPhoneAlarm[8] AND #SendDoneToVD THEN
       #Done[8] := TRUE;   // SR flip-flop
   END_IF;
   IF #InitDone[8] THEN #Done[8] := FALSE; END_IF;
END_REGION

REGION Network 48: **** 4.4 - Machine Status - Calculation **** Message Request Done
   // Message Request Done
   IF #VDReqPhoneAlarm[9] AND #SendDoneToVD THEN
       #Done[9] := TRUE;   // SR flip-flop
   END_IF;
   IF #InitDone[9] THEN #Done[9] := FALSE; END_IF;
END_REGION

REGION Network 49: **** 4.4 - Machine Status - Calculation **** Message Request Done
   // Message Request Done
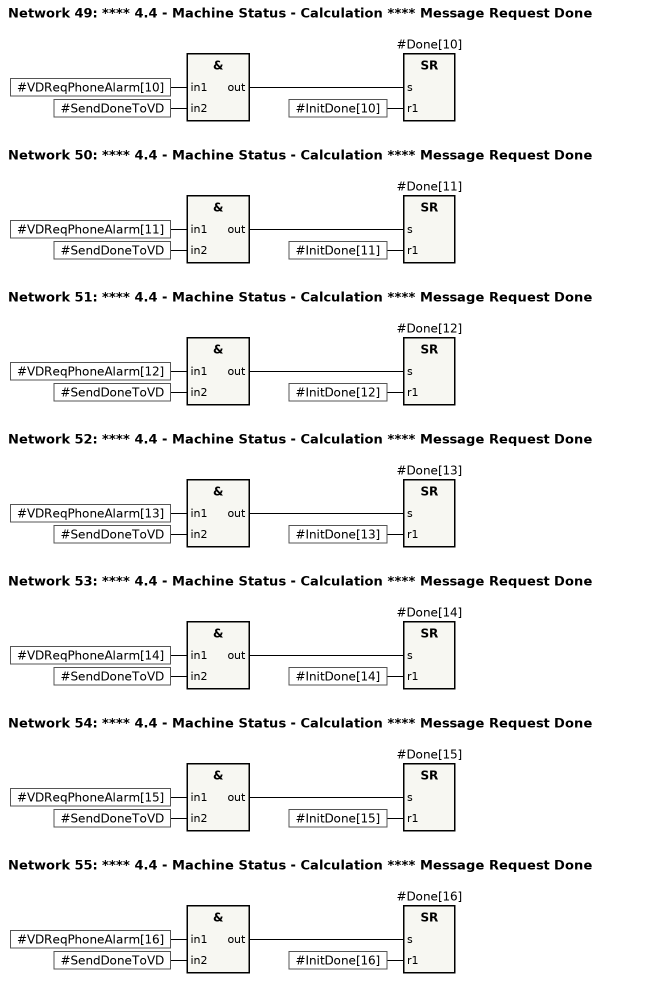
   IF #VDReqPhoneAlarm[10] AND #SendDoneToVD THEN
       #Done[10] := TRUE;   // SR flip-flop
   END_IF;
   IF #InitDone[10] THEN #Done[10] := FALSE; END_IF;
END_REGION

REGION Network 50: **** 4.4 - Machine Status - Calculation **** Message Request Done
   // Message Request Done
   IF #VDReqPhoneAlarm[11] AND #SendDoneToVD THEN
       #Done[11] := TRUE;   // SR flip-flop
   END_IF;
   IF #InitDone[11] THEN #Done[11] := FALSE; END_IF;
END_REGION

REGION Network 51: **** 4.4 - Machine Status - Calculation **** Message Request Done
   // Message Request Done
   IF #VDReqPhoneAlarm[12] AND #SendDoneToVD THEN
       #Done[12] := TRUE;   // SR flip-flop
   END_IF;
   IF #InitDone[12] THEN #Done[12] := FALSE; END_IF;
END_REGION

REGION Network 52: **** 4.4 - Machine Status - Calculation **** Message Request Done
   // Message Request Done
   IF #VDReqPhoneAlarm[13] AND #SendDoneToVD THEN
       #Done[13] := TRUE;   // SR flip-flop
   END_IF;
   IF #InitDone[13] THEN #Done[13] := FALSE; END_IF;
END_REGION

REGION Network 53: **** 4.4 - Machine Status - Calculation **** Message Request Done
   // Message Request Done
   IF #VDReqPhoneAlarm[14] AND #SendDoneToVD THEN
       #Done[14] := TRUE;   // SR flip-flop
   END_IF;
   IF #InitDone[14] THEN #Done[14] := FALSE; END_IF;
END_REGION

REGION Network 54: **** 4.4 - Machine Status - Calculation **** Message Request Done
   // Message Request Done
   IF #VDReqPhoneAlarm[15] AND #SendDoneToVD THEN
       #Done[15] := TRUE;   // SR flip-flop
   END_IF;
   IF #InitDone[15] THEN #Done[15] := FALSE; END_IF;
END_REGION

REGION Network 55: **** 4.4 - Machine Status - Calculation **** Message Request Done
   // Message Request Done
   IF #VDReqPhoneAlarm[16] AND #SendDoneToVD THEN
       #Done[16] := TRUE;   // SR flip-flop
   END_IF;
   IF #InitDone[16] THEN #Done[16] := FALSE; END_IF;
END_REGION

REGION Network 56: **** 4.4 - Machine Status - Calculation **** Que Message Request 1 / **** 4.4 - Machine Status - Calculation **** Queue Message Request 1
   // Que Message Request 1 / Queue Message Request 1
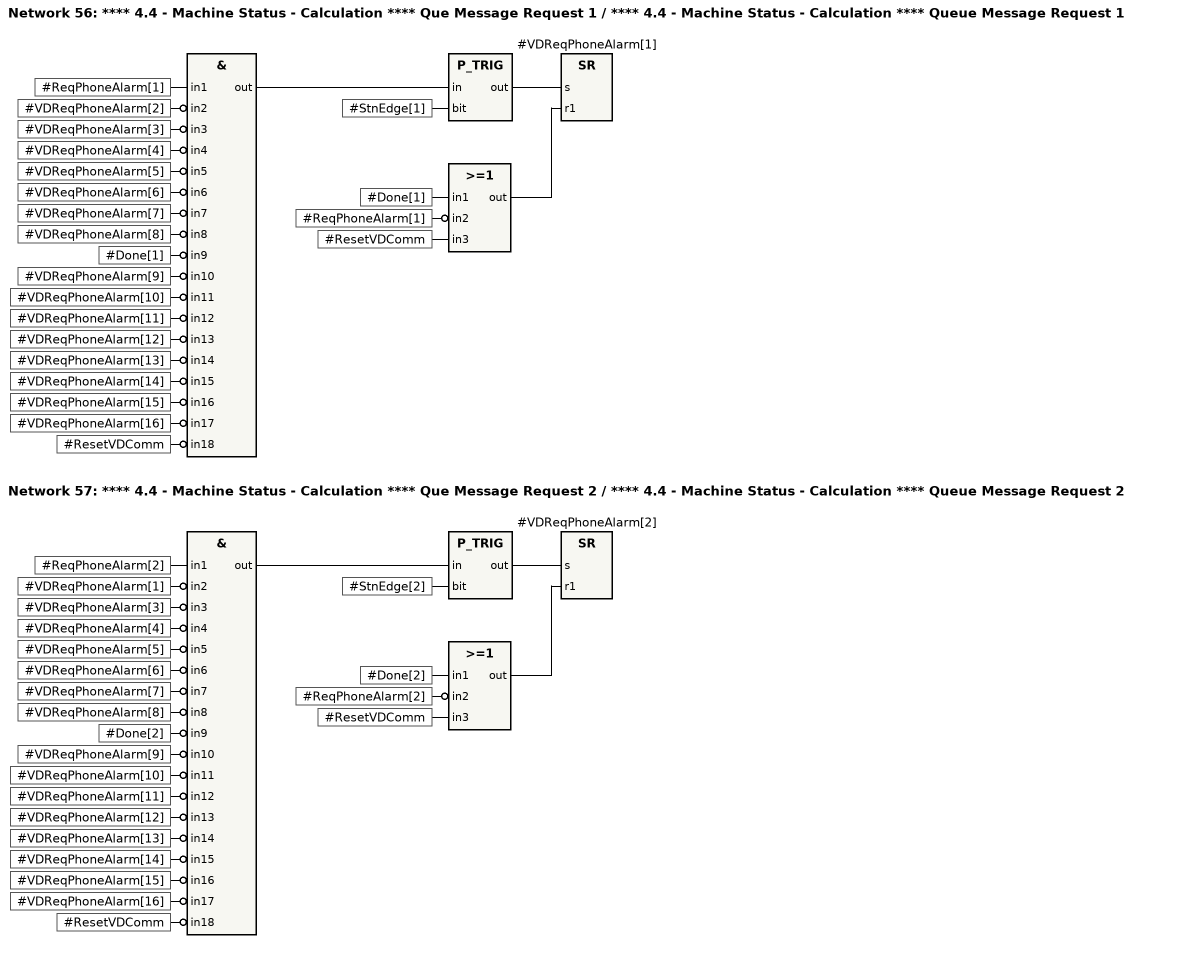
   #_w1 := #ReqPhoneAlarm[1] AND NOT #VDReqPhoneAlarm[2] AND NOT #VDReqPhoneAlarm[3] AND NOT #VDReqPhoneAlarm[4] AND NOT #VDReqPhoneAlarm[5] AND NOT #VDReqPhoneAlarm[6] AND NOT #VDReqPhoneAlarm[7] AND NOT #VDReqPhoneAlarm[8] AND NOT #Done[1] AND NOT #VDReqPhoneAlarm[9] AND NOT #VDReqPhoneAlarm[10] AND NOT #VDReqPhoneAlarm[11] AND NOT #VDReqPhoneAlarm[12] AND NOT #VDReqPhoneAlarm[13] AND NOT #VDReqPhoneAlarm[14] AND NOT #VDReqPhoneAlarm[15] AND NOT #VDReqPhoneAlarm[16] AND NOT #ResetVDComm;
   #_w2 := #_w1 AND NOT #StnEdge[1];   // rising edge
   #StnEdge[1] := #_w1;
   IF #_w2 THEN
       #VDReqPhoneAlarm[1] := TRUE;   // SR flip-flop
   END_IF;
   IF #Done[1] OR NOT #ReqPhoneAlarm[1] OR #ResetVDComm THEN #VDReqPhoneAlarm[1] := FALSE; END_IF;
END_REGION

REGION Network 57: **** 4.4 - Machine Status - Calculation **** Que Message Request 2 / **** 4.4 - Machine Status - Calculation **** Queue Message Request 2
   // Que Message Request 2 / Queue Message Request 2
   #_w1 := #ReqPhoneAlarm[2] AND NOT #VDReqPhoneAlarm[1] AND NOT #VDReqPhoneAlarm[3] AND NOT #VDReqPhoneAlarm[4] AND NOT #VDReqPhoneAlarm[5] AND NOT #VDReqPhoneAlarm[6] AND NOT #VDReqPhoneAlarm[7] AND NOT #VDReqPhoneAlarm[8] AND NOT #Done[2] AND NOT #VDReqPhoneAlarm[9] AND NOT #VDReqPhoneAlarm[10] AND NOT #VDReqPhoneAlarm[11] AND NOT #VDReqPhoneAlarm[12] AND NOT #VDReqPhoneAlarm[13] AND NOT #VDReqPhoneAlarm[14] AND NOT #VDReqPhoneAlarm[15] AND NOT #VDReqPhoneAlarm[16] AND NOT #ResetVDComm;
   #_w2 := #_w1 AND NOT #StnEdge[2];   // rising edge
   #StnEdge[2] := #_w1;
   IF #_w2 THEN
       #VDReqPhoneAlarm[2] := TRUE;   // SR flip-flop
   END_IF;
   IF #Done[2] OR NOT #ReqPhoneAlarm[2] OR #ResetVDComm THEN #VDReqPhoneAlarm[2] := FALSE; END_IF;
END_REGION

REGION Network 58: **** 4.4 - Machine Status - Calculation **** Que Message Request 3 / **** 4.4 - Machine Status - Calculation **** Queue Message Request 3
   // Que Message Request 3 / Queue Message Request 3
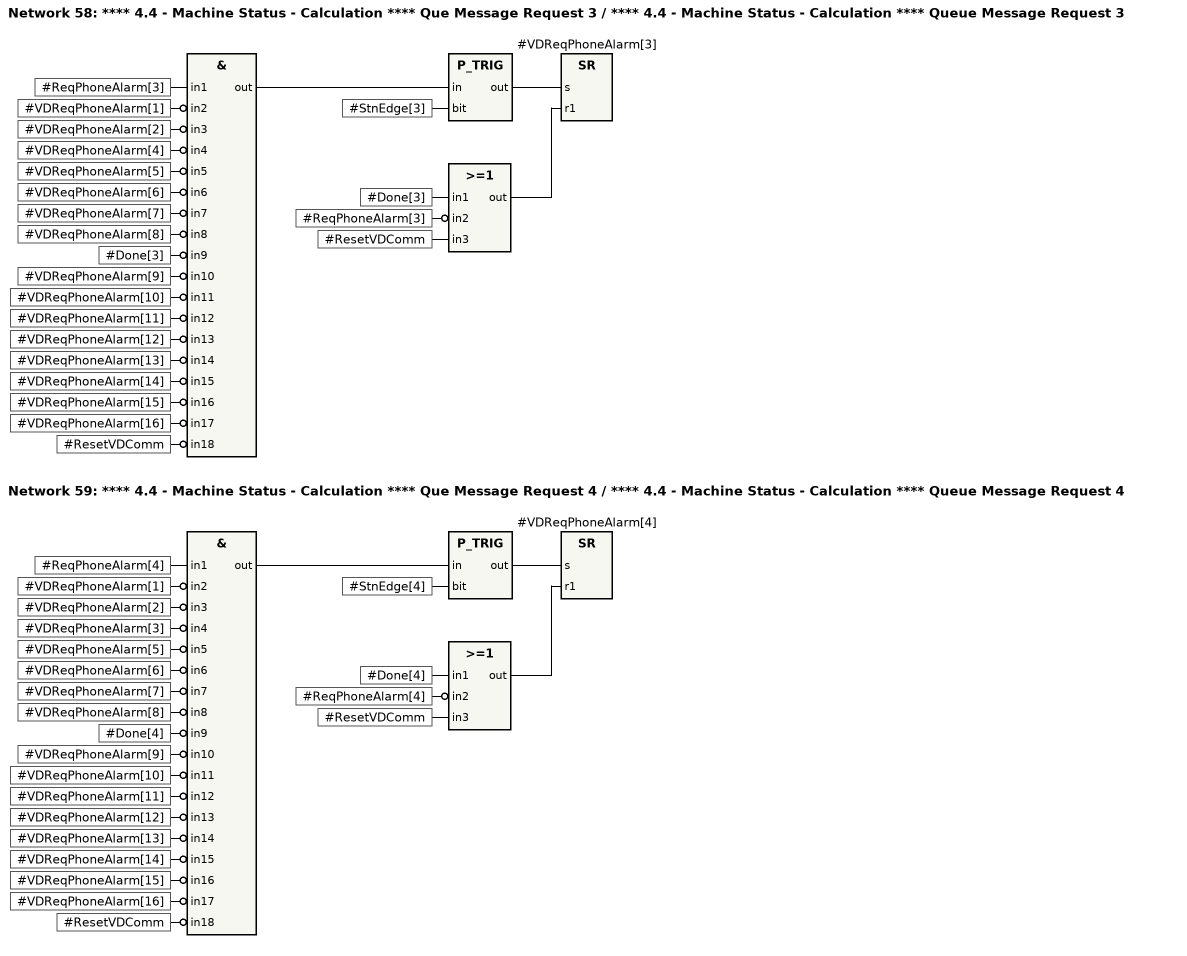
   #_w1 := #ReqPhoneAlarm[3] AND NOT #VDReqPhoneAlarm[1] AND NOT #VDReqPhoneAlarm[2] AND NOT #VDReqPhoneAlarm[4] AND NOT #VDReqPhoneAlarm[5] AND NOT #VDReqPhoneAlarm[6] AND NOT #VDReqPhoneAlarm[7] AND NOT #VDReqPhoneAlarm[8] AND NOT #Done[3] AND NOT #VDReqPhoneAlarm[9] AND NOT #VDReqPhoneAlarm[10] AND NOT #VDReqPhoneAlarm[11] AND NOT #VDReqPhoneAlarm[12] AND NOT #VDReqPhoneAlarm[13] AND NOT #VDReqPhoneAlarm[14] AND NOT #VDReqPhoneAlarm[15] AND NOT #VDReqPhoneAlarm[16] AND NOT #ResetVDComm;
   #_w2 := #_w1 AND NOT #StnEdge[3];   // rising edge
   #StnEdge[3] := #_w1;
   IF #_w2 THEN
       #VDReqPhoneAlarm[3] := TRUE;   // SR flip-flop
   END_IF;
   IF #Done[3] OR NOT #ReqPhoneAlarm[3] OR #ResetVDComm THEN #VDReqPhoneAlarm[3] := FALSE; END_IF;
END_REGION

REGION Network 59: **** 4.4 - Machine Status - Calculation **** Que Message Request 4 / **** 4.4 - Machine Status - Calculation **** Queue Message Request 4
   // Que Message Request 4 / Queue Message Request 4
   #_w1 := #ReqPhoneAlarm[4] AND NOT #VDReqPhoneAlarm[1] AND NOT #VDReqPhoneAlarm[2] AND NOT #VDReqPhoneAlarm[3] AND NOT #VDReqPhoneAlarm[5] AND NOT #VDReqPhoneAlarm[6] AND NOT #VDReqPhoneAlarm[7] AND NOT #VDReqPhoneAlarm[8] AND NOT #Done[4] AND NOT #VDReqPhoneAlarm[9] AND NOT #VDReqPhoneAlarm[10] AND NOT #VDReqPhoneAlarm[11] AND NOT #VDReqPhoneAlarm[12] AND NOT #VDReqPhoneAlarm[13] AND NOT #VDReqPhoneAlarm[14] AND NOT #VDReqPhoneAlarm[15] AND NOT #VDReqPhoneAlarm[16] AND NOT #ResetVDComm;
   #_w2 := #_w1 AND NOT #StnEdge[4];   // rising edge
   #StnEdge[4] := #_w1;
   IF #_w2 THEN
       #VDReqPhoneAlarm[4] := TRUE;   // SR flip-flop
   END_IF;
   IF #Done[4] OR NOT #ReqPhoneAlarm[4] OR #ResetVDComm THEN #VDReqPhoneAlarm[4] := FALSE; END_IF;
END_REGION

REGION Network 60: **** 4.4 - Machine Status - Calculation **** Que Message Request 5 / **** 4.4 - Machine Status - Calculation **** Queue Message Request 5
   // Que Message Request 5 / Queue Message Request 5
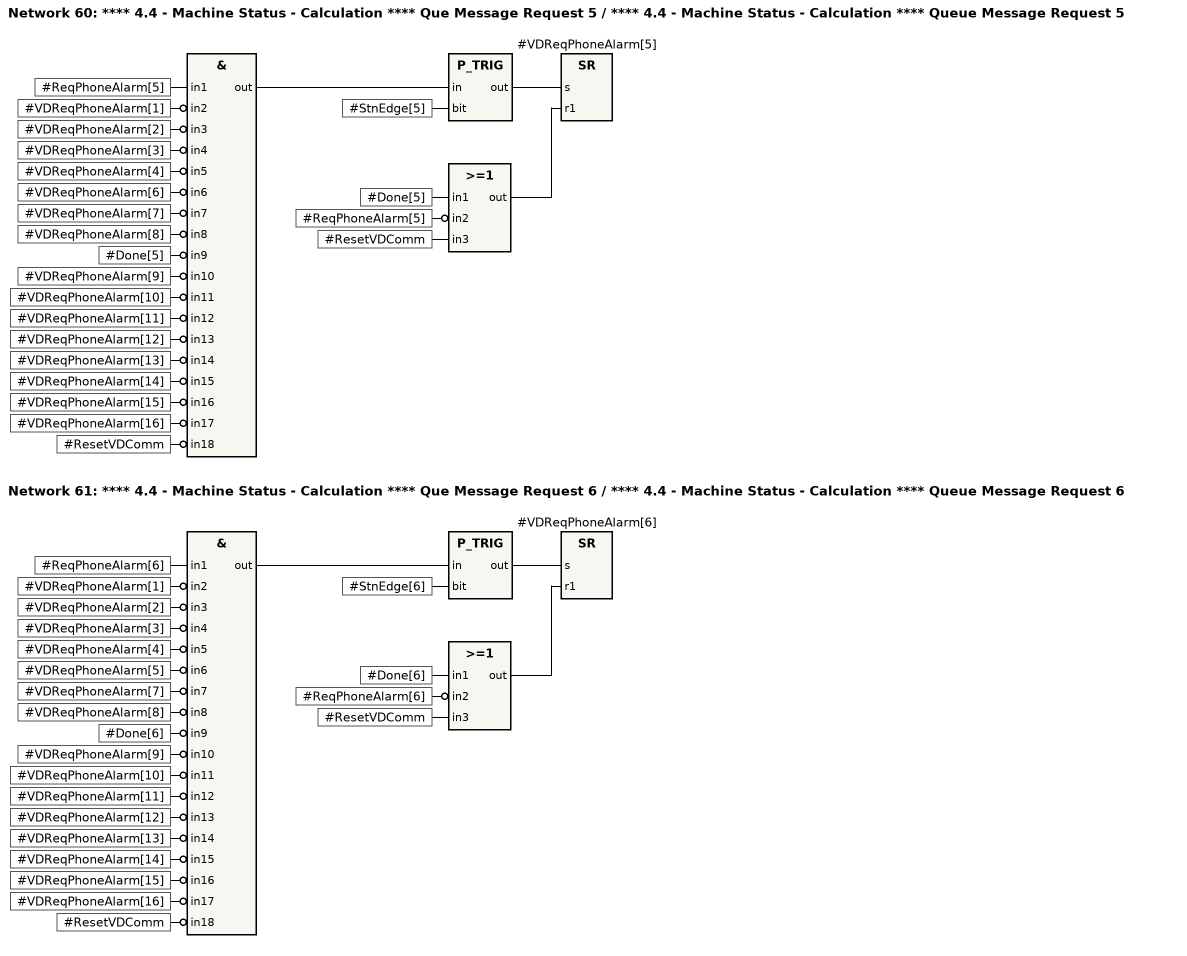
   #_w1 := #ReqPhoneAlarm[5] AND NOT #VDReqPhoneAlarm[1] AND NOT #VDReqPhoneAlarm[2] AND NOT #VDReqPhoneAlarm[3] AND NOT #VDReqPhoneAlarm[4] AND NOT #VDReqPhoneAlarm[6] AND NOT #VDReqPhoneAlarm[7] AND NOT #VDReqPhoneAlarm[8] AND NOT #Done[5] AND NOT #VDReqPhoneAlarm[9] AND NOT #VDReqPhoneAlarm[10] AND NOT #VDReqPhoneAlarm[11] AND NOT #VDReqPhoneAlarm[12] AND NOT #VDReqPhoneAlarm[13] AND NOT #VDReqPhoneAlarm[14] AND NOT #VDReqPhoneAlarm[15] AND NOT #VDReqPhoneAlarm[16] AND NOT #ResetVDComm;
   #_w2 := #_w1 AND NOT #StnEdge[5];   // rising edge
   #StnEdge[5] := #_w1;
   IF #_w2 THEN
       #VDReqPhoneAlarm[5] := TRUE;   // SR flip-flop
   END_IF;
   IF #Done[5] OR NOT #ReqPhoneAlarm[5] OR #ResetVDComm THEN #VDReqPhoneAlarm[5] := FALSE; END_IF;
END_REGION

REGION Network 61: **** 4.4 - Machine Status - Calculation **** Que Message Request 6 / **** 4.4 - Machine Status - Calculation **** Queue Message Request 6
   // Que Message Request 6 / Queue Message Request 6
   #_w1 := #ReqPhoneAlarm[6] AND NOT #VDReqPhoneAlarm[1] AND NOT #VDReqPhoneAlarm[2] AND NOT #VDReqPhoneAlarm[3] AND NOT #VDReqPhoneAlarm[4] AND NOT #VDReqPhoneAlarm[5] AND NOT #VDReqPhoneAlarm[7] AND NOT #VDReqPhoneAlarm[8] AND NOT #Done[6] AND NOT #VDReqPhoneAlarm[9] AND NOT #VDReqPhoneAlarm[10] AND NOT #VDReqPhoneAlarm[11] AND NOT #VDReqPhoneAlarm[12] AND NOT #VDReqPhoneAlarm[13] AND NOT #VDReqPhoneAlarm[14] AND NOT #VDReqPhoneAlarm[15] AND NOT #VDReqPhoneAlarm[16] AND NOT #ResetVDComm;
   #_w2 := #_w1 AND NOT #StnEdge[6];   // rising edge
   #StnEdge[6] := #_w1;
   IF #_w2 THEN
       #VDReqPhoneAlarm[6] := TRUE;   // SR flip-flop
   END_IF;
   IF #Done[6] OR NOT #ReqPhoneAlarm[6] OR #ResetVDComm THEN #VDReqPhoneAlarm[6] := FALSE; END_IF;
END_REGION

REGION Network 62: **** 4.4 - Machine Status - Calculation **** Que Message Request 7 / **** 4.4 - Machine Status - Calculation **** Queue Message Request 7
   // Que Message Request 7 / Queue Message Request 7
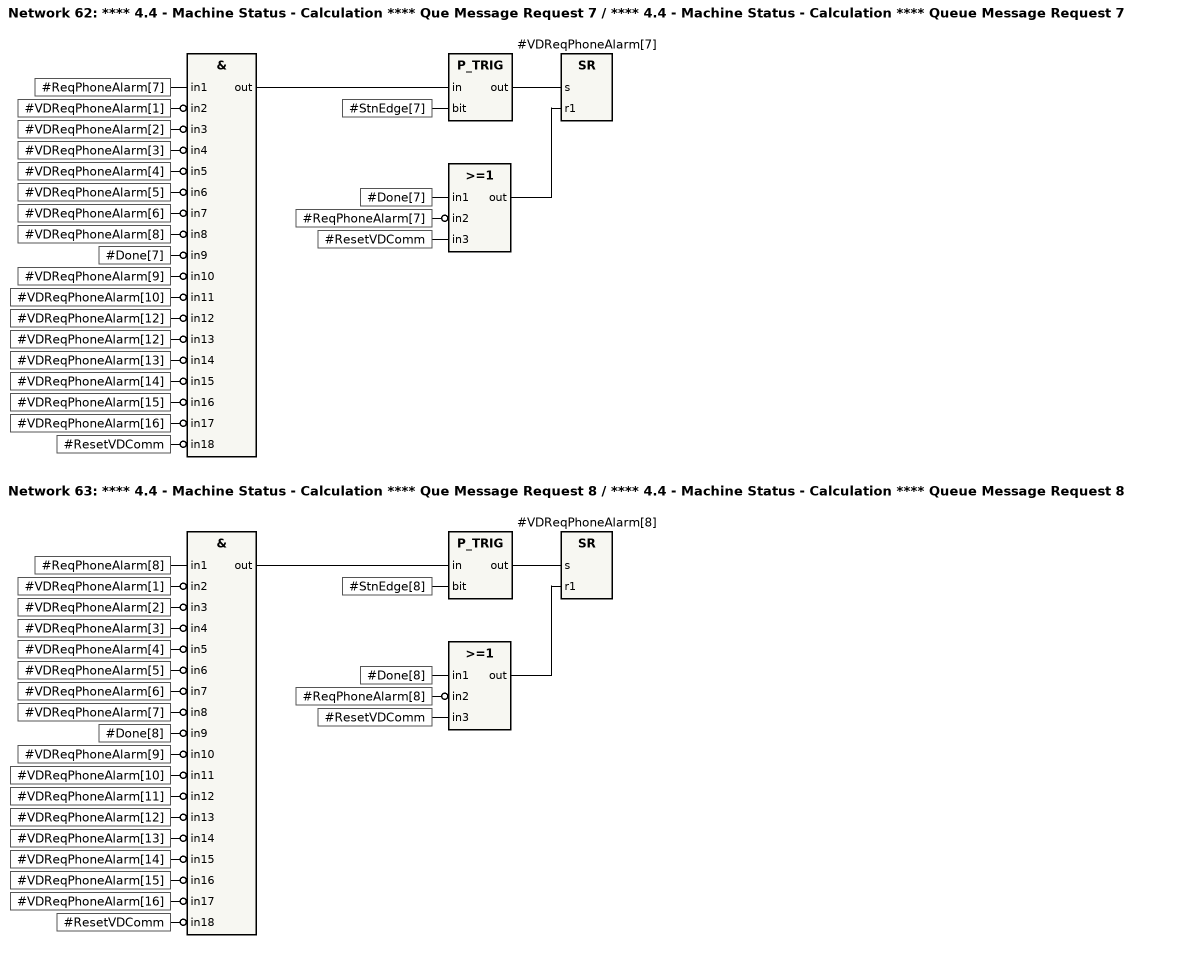
   #_w1 := #ReqPhoneAlarm[7] AND NOT #VDReqPhoneAlarm[1] AND NOT #VDReqPhoneAlarm[2] AND NOT #VDReqPhoneAlarm[3] AND NOT #VDReqPhoneAlarm[4] AND NOT #VDReqPhoneAlarm[5] AND NOT #VDReqPhoneAlarm[6] AND NOT #VDReqPhoneAlarm[8] AND NOT #Done[7] AND NOT #VDReqPhoneAlarm[9] AND NOT #VDReqPhoneAlarm[10] AND NOT #VDReqPhoneAlarm[12] AND NOT #VDReqPhoneAlarm[12] AND NOT #VDReqPhoneAlarm[13] AND NOT #VDReqPhoneAlarm[14] AND NOT #VDReqPhoneAlarm[15] AND NOT #VDReqPhoneAlarm[16] AND NOT #ResetVDComm;
   #_w2 := #_w1 AND NOT #StnEdge[7];   // rising edge
   #StnEdge[7] := #_w1;
   IF #_w2 THEN
       #VDReqPhoneAlarm[7] := TRUE;   // SR flip-flop
   END_IF;
   IF #Done[7] OR NOT #ReqPhoneAlarm[7] OR #ResetVDComm THEN #VDReqPhoneAlarm[7] := FALSE; END_IF;
END_REGION

REGION Network 63: **** 4.4 - Machine Status - Calculation **** Que Message Request 8 / **** 4.4 - Machine Status - Calculation **** Queue Message Request 8
   // Que Message Request 8 / Queue Message Request 8
   #_w1 := #ReqPhoneAlarm[8] AND NOT #VDReqPhoneAlarm[1] AND NOT #VDReqPhoneAlarm[2] AND NOT #VDReqPhoneAlarm[3] AND NOT #VDReqPhoneAlarm[4] AND NOT #VDReqPhoneAlarm[5] AND NOT #VDReqPhoneAlarm[6] AND NOT #VDReqPhoneAlarm[7] AND NOT #Done[8] AND NOT #VDReqPhoneAlarm[9] AND NOT #VDReqPhoneAlarm[10] AND NOT #VDReqPhoneAlarm[11] AND NOT #VDReqPhoneAlarm[12] AND NOT #VDReqPhoneAlarm[13] AND NOT #VDReqPhoneAlarm[14] AND NOT #VDReqPhoneAlarm[15] AND NOT #VDReqPhoneAlarm[16] AND NOT #ResetVDComm;
   #_w2 := #_w1 AND NOT #StnEdge[8];   // rising edge
   #StnEdge[8] := #_w1;
   IF #_w2 THEN
       #VDReqPhoneAlarm[8] := TRUE;   // SR flip-flop
   END_IF;
   IF #Done[8] OR NOT #ReqPhoneAlarm[8] OR #ResetVDComm THEN #VDReqPhoneAlarm[8] := FALSE; END_IF;
END_REGION

REGION Network 64: **** 4.4 - Machine Status - Calculation **** Que Message Request 9 / **** 4.4 - Machine Status - Calculation **** Queue Message Request 9
   // Que Message Request 9 / Queue Message Request 9
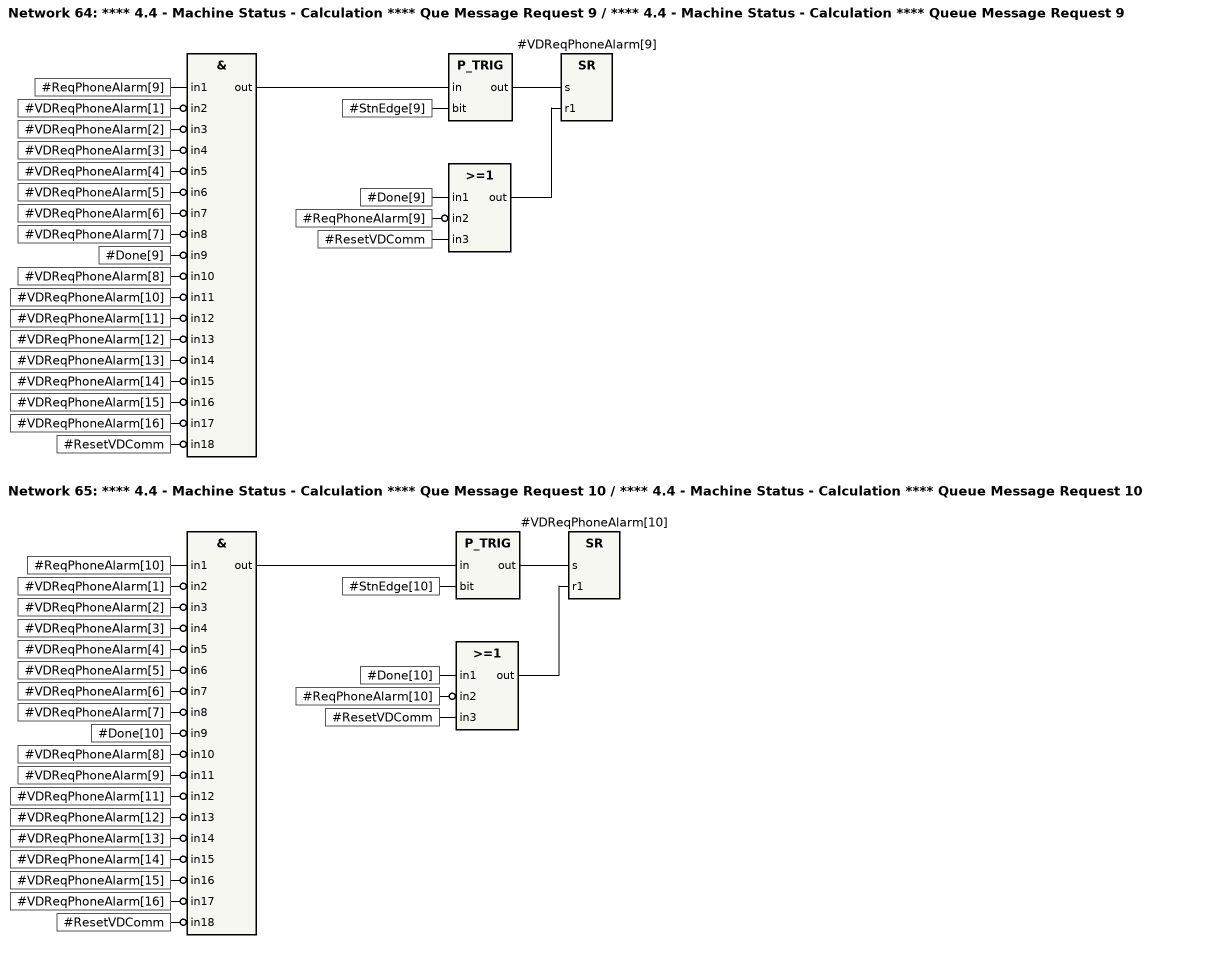
   #_w1 := #ReqPhoneAlarm[9] AND NOT #VDReqPhoneAlarm[1] AND NOT #VDReqPhoneAlarm[2] AND NOT #VDReqPhoneAlarm[3] AND NOT #VDReqPhoneAlarm[4] AND NOT #VDReqPhoneAlarm[5] AND NOT #VDReqPhoneAlarm[6] AND NOT #VDReqPhoneAlarm[7] AND NOT #Done[9] AND NOT #VDReqPhoneAlarm[8] AND NOT #VDReqPhoneAlarm[10] AND NOT #VDReqPhoneAlarm[11] AND NOT #VDReqPhoneAlarm[12] AND NOT #VDReqPhoneAlarm[13] AND NOT #VDReqPhoneAlarm[14] AND NOT #VDReqPhoneAlarm[15] AND NOT #VDReqPhoneAlarm[16] AND NOT #ResetVDComm;
   #_w2 := #_w1 AND NOT #StnEdge[9];   // rising edge
   #StnEdge[9] := #_w1;
   IF #_w2 THEN
       #VDReqPhoneAlarm[9] := TRUE;   // SR flip-flop
   END_IF;
   IF #Done[9] OR NOT #ReqPhoneAlarm[9] OR #ResetVDComm THEN #VDReqPhoneAlarm[9] := FALSE; END_IF;
END_REGION

REGION Network 65: **** 4.4 - Machine Status - Calculation **** Que Message Request 10 / **** 4.4 - Machine Status - Calculation **** Queue Message Request 10
   // Que Message Request 10 / Queue Message Request 10
   #_w1 := #ReqPhoneAlarm[10] AND NOT #VDReqPhoneAlarm[1] AND NOT #VDReqPhoneAlarm[2] AND NOT #VDReqPhoneAlarm[3] AND NOT #VDReqPhoneAlarm[4] AND NOT #VDReqPhoneAlarm[5] AND NOT #VDReqPhoneAlarm[6] AND NOT #VDReqPhoneAlarm[7] AND NOT #Done[10] AND NOT #VDReqPhoneAlarm[8] AND NOT #VDReqPhoneAlarm[9] AND NOT #VDReqPhoneAlarm[11] AND NOT #VDReqPhoneAlarm[12] AND NOT #VDReqPhoneAlarm[13] AND NOT #VDReqPhoneAlarm[14] AND NOT #VDReqPhoneAlarm[15] AND NOT #VDReqPhoneAlarm[16] AND NOT #ResetVDComm;
   #_w2 := #_w1 AND NOT #StnEdge[10];   // rising edge
   #StnEdge[10] := #_w1;
   IF #_w2 THEN
       #VDReqPhoneAlarm[10] := TRUE;   // SR flip-flop
   END_IF;
   IF #Done[10] OR NOT #ReqPhoneAlarm[10] OR #ResetVDComm THEN #VDReqPhoneAlarm[10] := FALSE; END_IF;
END_REGION

REGION Network 66: **** 4.4 - Machine Status - Calculation **** Que Message Request 11 / **** 4.4 - Machine Status - Calculation **** Queue Message Request 11
   // Que Message Request 11 / Queue Message Request 11
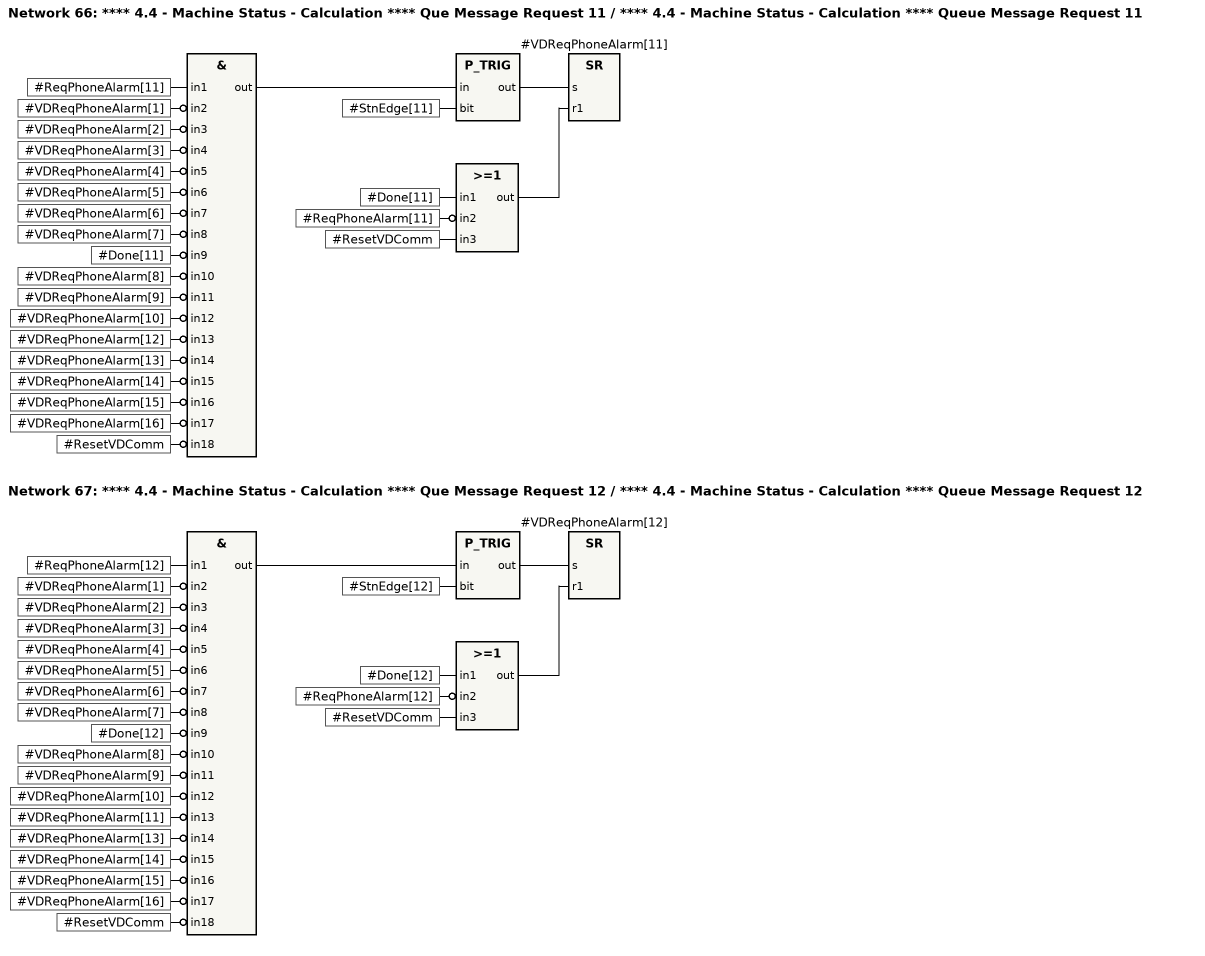
   #_w1 := #ReqPhoneAlarm[11] AND NOT #VDReqPhoneAlarm[1] AND NOT #VDReqPhoneAlarm[2] AND NOT #VDReqPhoneAlarm[3] AND NOT #VDReqPhoneAlarm[4] AND NOT #VDReqPhoneAlarm[5] AND NOT #VDReqPhoneAlarm[6] AND NOT #VDReqPhoneAlarm[7] AND NOT #Done[11] AND NOT #VDReqPhoneAlarm[8] AND NOT #VDReqPhoneAlarm[9] AND NOT #VDReqPhoneAlarm[10] AND NOT #VDReqPhoneAlarm[12] AND NOT #VDReqPhoneAlarm[13] AND NOT #VDReqPhoneAlarm[14] AND NOT #VDReqPhoneAlarm[15] AND NOT #VDReqPhoneAlarm[16] AND NOT #ResetVDComm;
   #_w2 := #_w1 AND NOT #StnEdge[11];   // rising edge
   #StnEdge[11] := #_w1;
   IF #_w2 THEN
       #VDReqPhoneAlarm[11] := TRUE;   // SR flip-flop
   END_IF;
   IF #Done[11] OR NOT #ReqPhoneAlarm[11] OR #ResetVDComm THEN #VDReqPhoneAlarm[11] := FALSE; END_IF;
END_REGION

REGION Network 67: **** 4.4 - Machine Status - Calculation **** Que Message Request 12 / **** 4.4 - Machine Status - Calculation **** Queue Message Request 12
   // Que Message Request 12 / Queue Message Request 12
   #_w1 := #ReqPhoneAlarm[12] AND NOT #VDReqPhoneAlarm[1] AND NOT #VDReqPhoneAlarm[2] AND NOT #VDReqPhoneAlarm[3] AND NOT #VDReqPhoneAlarm[4] AND NOT #VDReqPhoneAlarm[5] AND NOT #VDReqPhoneAlarm[6] AND NOT #VDReqPhoneAlarm[7] AND NOT #Done[12] AND NOT #VDReqPhoneAlarm[8] AND NOT #VDReqPhoneAlarm[9] AND NOT #VDReqPhoneAlarm[10] AND NOT #VDReqPhoneAlarm[11] AND NOT #VDReqPhoneAlarm[13] AND NOT #VDReqPhoneAlarm[14] AND NOT #VDReqPhoneAlarm[15] AND NOT #VDReqPhoneAlarm[16] AND NOT #ResetVDComm;
   #_w2 := #_w1 AND NOT #StnEdge[12];   // rising edge
   #StnEdge[12] := #_w1;
   IF #_w2 THEN
       #VDReqPhoneAlarm[12] := TRUE;   // SR flip-flop
   END_IF;
   IF #Done[12] OR NOT #ReqPhoneAlarm[12] OR #ResetVDComm THEN #VDReqPhoneAlarm[12] := FALSE; END_IF;
END_REGION

REGION Network 68: **** 4.4 - Machine Status - Calculation **** Que Message Request 13 / **** 4.4 - Machine Status - Calculation **** Queue Message Request 13
   // Que Message Request 13 / Queue Message Request 13
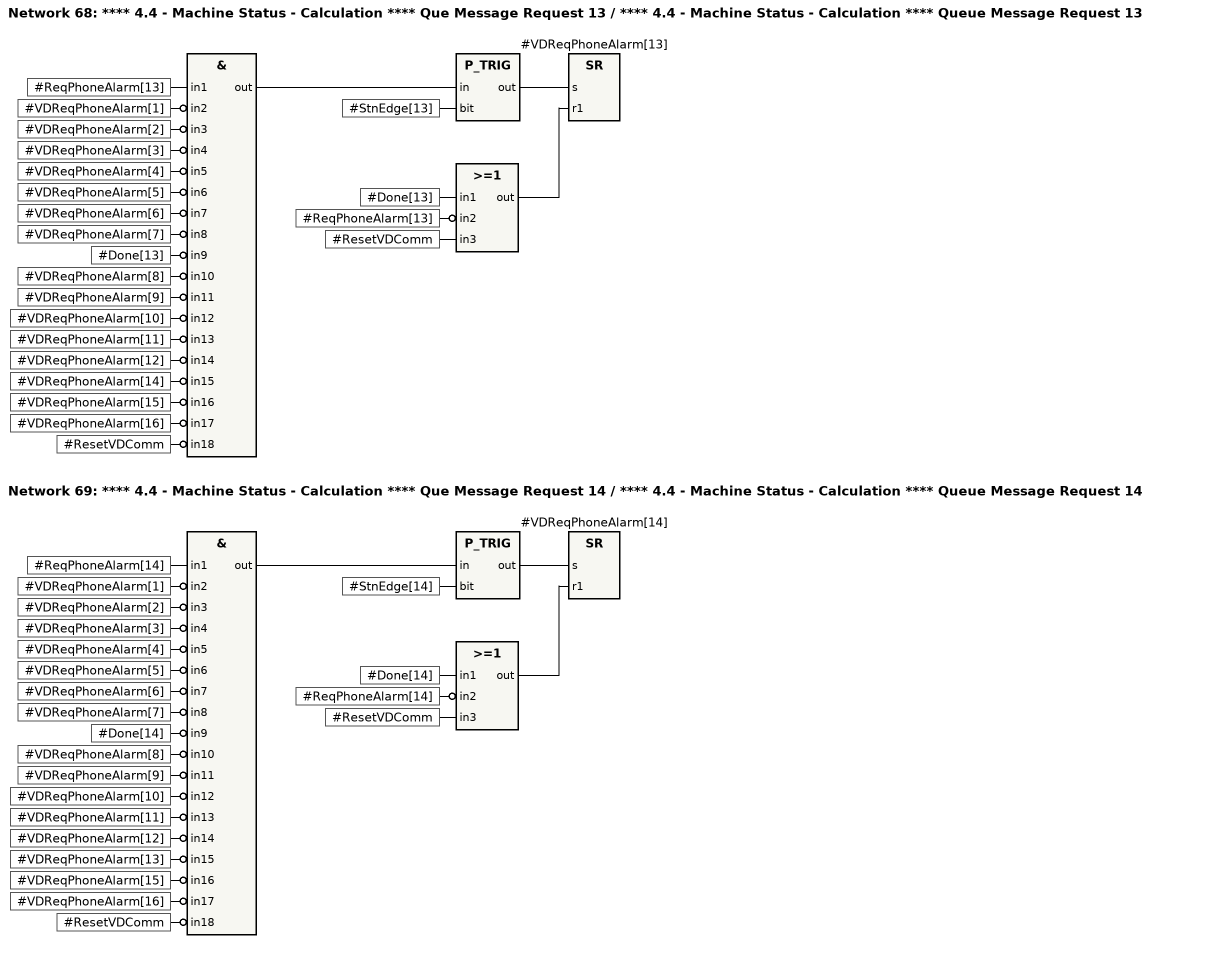
   #_w1 := #ReqPhoneAlarm[13] AND NOT #VDReqPhoneAlarm[1] AND NOT #VDReqPhoneAlarm[2] AND NOT #VDReqPhoneAlarm[3] AND NOT #VDReqPhoneAlarm[4] AND NOT #VDReqPhoneAlarm[5] AND NOT #VDReqPhoneAlarm[6] AND NOT #VDReqPhoneAlarm[7] AND NOT #Done[13] AND NOT #VDReqPhoneAlarm[8] AND NOT #VDReqPhoneAlarm[9] AND NOT #VDReqPhoneAlarm[10] AND NOT #VDReqPhoneAlarm[11] AND NOT #VDReqPhoneAlarm[12] AND NOT #VDReqPhoneAlarm[14] AND NOT #VDReqPhoneAlarm[15] AND NOT #VDReqPhoneAlarm[16] AND NOT #ResetVDComm;
   #_w2 := #_w1 AND NOT #StnEdge[13];   // rising edge
   #StnEdge[13] := #_w1;
   IF #_w2 THEN
       #VDReqPhoneAlarm[13] := TRUE;   // SR flip-flop
   END_IF;
   IF #Done[13] OR NOT #ReqPhoneAlarm[13] OR #ResetVDComm THEN #VDReqPhoneAlarm[13] := FALSE; END_IF;
END_REGION

REGION Network 69: **** 4.4 - Machine Status - Calculation **** Que Message Request 14 / **** 4.4 - Machine Status - Calculation **** Queue Message Request 14
   // Que Message Request 14 / Queue Message Request 14
   #_w1 := #ReqPhoneAlarm[14] AND NOT #VDReqPhoneAlarm[1] AND NOT #VDReqPhoneAlarm[2] AND NOT #VDReqPhoneAlarm[3] AND NOT #VDReqPhoneAlarm[4] AND NOT #VDReqPhoneAlarm[5] AND NOT #VDReqPhoneAlarm[6] AND NOT #VDReqPhoneAlarm[7] AND NOT #Done[14] AND NOT #VDReqPhoneAlarm[8] AND NOT #VDReqPhoneAlarm[9] AND NOT #VDReqPhoneAlarm[10] AND NOT #VDReqPhoneAlarm[11] AND NOT #VDReqPhoneAlarm[12] AND NOT #VDReqPhoneAlarm[13] AND NOT #VDReqPhoneAlarm[15] AND NOT #VDReqPhoneAlarm[16] AND NOT #ResetVDComm;
   #_w2 := #_w1 AND NOT #StnEdge[14];   // rising edge
   #StnEdge[14] := #_w1;
   IF #_w2 THEN
       #VDReqPhoneAlarm[14] := TRUE;   // SR flip-flop
   END_IF;
   IF #Done[14] OR NOT #ReqPhoneAlarm[14] OR #ResetVDComm THEN #VDReqPhoneAlarm[14] := FALSE; END_IF;
END_REGION

REGION Network 70: **** 4.4 - Machine Status - Calculation **** Que Message Request 15 / **** 4.4 - Machine Status - Calculation **** Queue Message Request 15
   // Que Message Request 15 / Queue Message Request 15
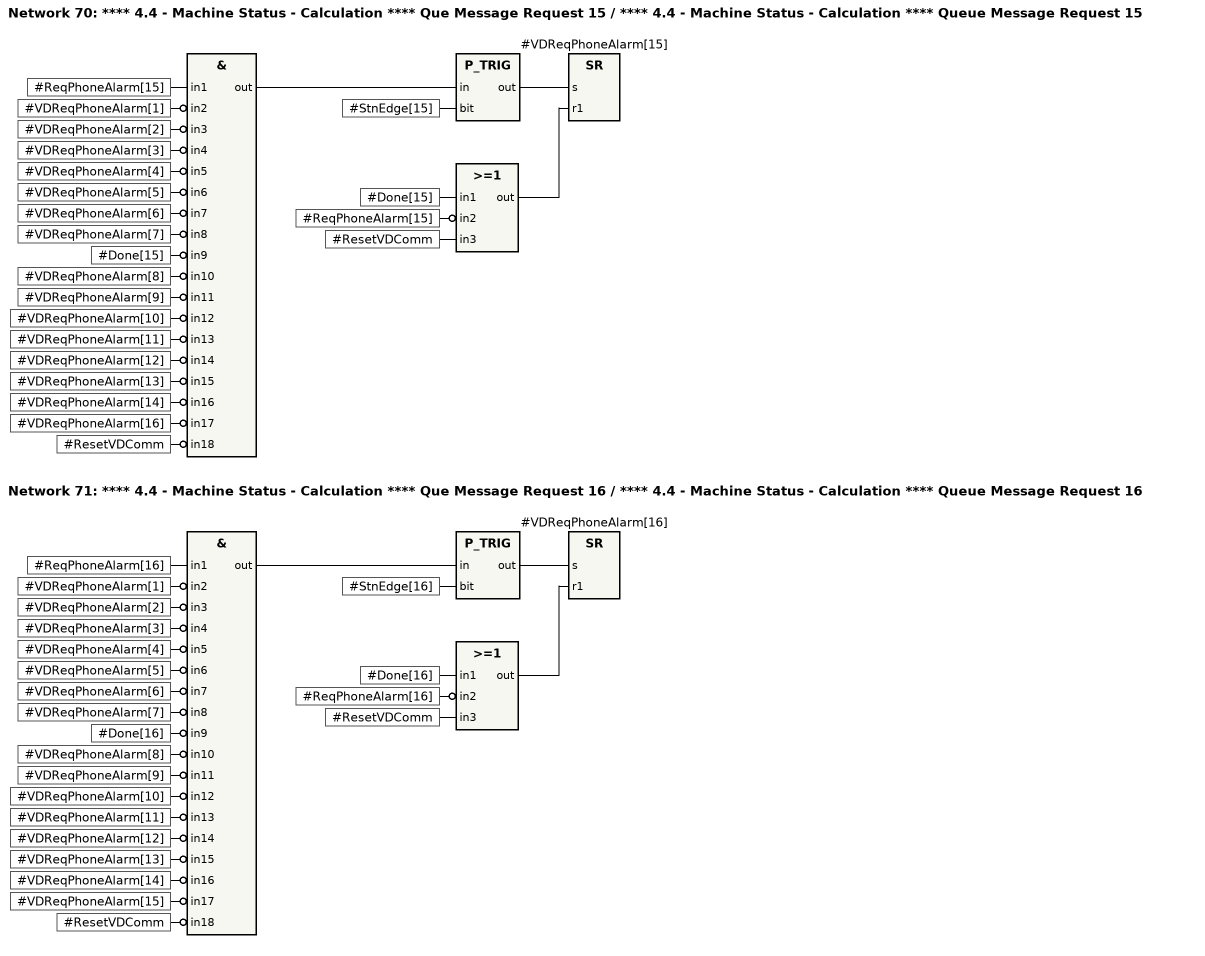
   #_w1 := #ReqPhoneAlarm[15] AND NOT #VDReqPhoneAlarm[1] AND NOT #VDReqPhoneAlarm[2] AND NOT #VDReqPhoneAlarm[3] AND NOT #VDReqPhoneAlarm[4] AND NOT #VDReqPhoneAlarm[5] AND NOT #VDReqPhoneAlarm[6] AND NOT #VDReqPhoneAlarm[7] AND NOT #Done[15] AND NOT #VDReqPhoneAlarm[8] AND NOT #VDReqPhoneAlarm[9] AND NOT #VDReqPhoneAlarm[10] AND NOT #VDReqPhoneAlarm[11] AND NOT #VDReqPhoneAlarm[12] AND NOT #VDReqPhoneAlarm[13] AND NOT #VDReqPhoneAlarm[14] AND NOT #VDReqPhoneAlarm[16] AND NOT #ResetVDComm;
   #_w2 := #_w1 AND NOT #StnEdge[15];   // rising edge
   #StnEdge[15] := #_w1;
   IF #_w2 THEN
       #VDReqPhoneAlarm[15] := TRUE;   // SR flip-flop
   END_IF;
   IF #Done[15] OR NOT #ReqPhoneAlarm[15] OR #ResetVDComm THEN #VDReqPhoneAlarm[15] := FALSE; END_IF;
END_REGION

REGION Network 71: **** 4.4 - Machine Status - Calculation **** Que Message Request 16 / **** 4.4 - Machine Status - Calculation **** Queue Message Request 16
   // Que Message Request 16 / Queue Message Request 16
   #_w1 := #ReqPhoneAlarm[16] AND NOT #VDReqPhoneAlarm[1] AND NOT #VDReqPhoneAlarm[2] AND NOT #VDReqPhoneAlarm[3] AND NOT #VDReqPhoneAlarm[4] AND NOT #VDReqPhoneAlarm[5] AND NOT #VDReqPhoneAlarm[6] AND NOT #VDReqPhoneAlarm[7] AND NOT #Done[16] AND NOT #VDReqPhoneAlarm[8] AND NOT #VDReqPhoneAlarm[9] AND NOT #VDReqPhoneAlarm[10] AND NOT #VDReqPhoneAlarm[11] AND NOT #VDReqPhoneAlarm[12] AND NOT #VDReqPhoneAlarm[13] AND NOT #VDReqPhoneAlarm[14] AND NOT #VDReqPhoneAlarm[15] AND NOT #ResetVDComm;
   #_w2 := #_w1 AND NOT #StnEdge[16];   // rising edge
   #StnEdge[16] := #_w1;
   IF #_w2 THEN
       #VDReqPhoneAlarm[16] := TRUE;   // SR flip-flop
   END_IF;
   IF #Done[16] OR NOT #ReqPhoneAlarm[16] OR #ResetVDComm THEN #VDReqPhoneAlarm[16] := FALSE; END_IF;
END_REGION

REGION Network 72: **** 4.6 - Machine status - Indication **** Animation / **** 4.6 - Machine status - Indication **** Animation SP1
   // Animation
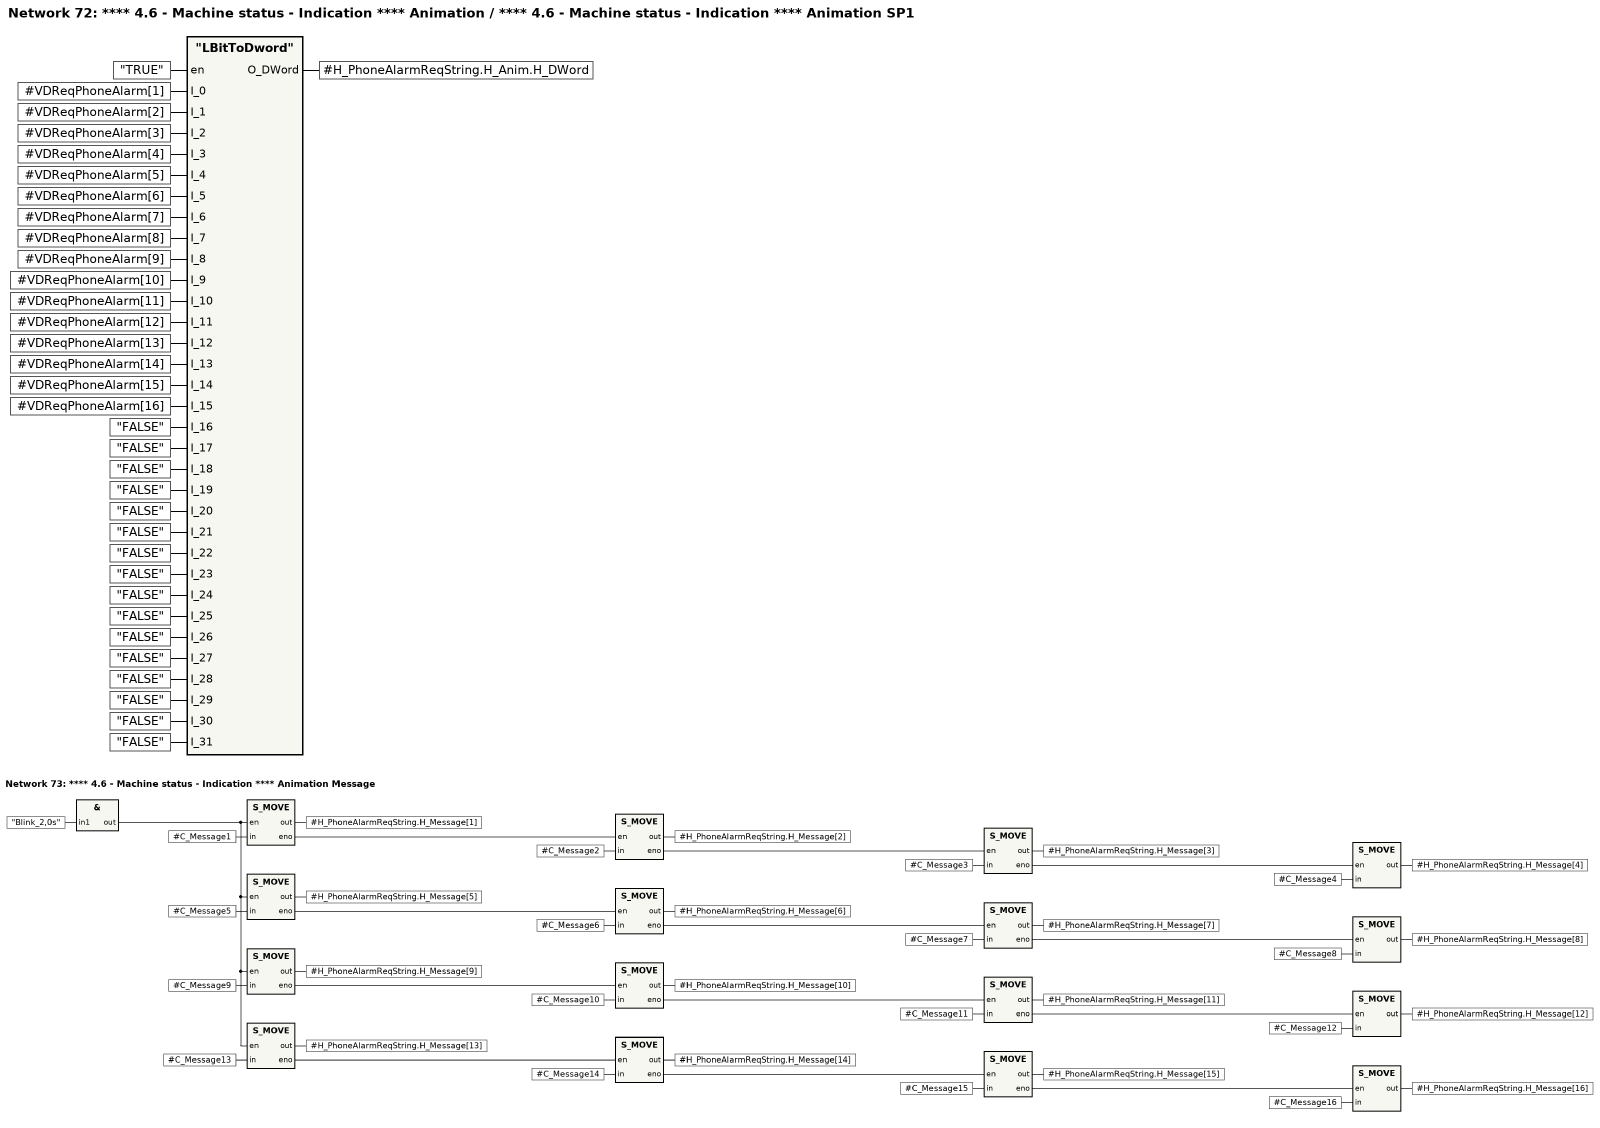
   IF "TRUE" THEN
       "LBitToDword"(I_0 := #VDReqPhoneAlarm[1],
                     I_1 := #VDReqPhoneAlarm[2],
                     I_2 := #VDReqPhoneAlarm[3],
                     I_3 := #VDReqPhoneAlarm[4],
                     I_4 := #VDReqPhoneAlarm[5],
                     I_5 := #VDReqPhoneAlarm[6],
                     I_6 := #VDReqPhoneAlarm[7],
                     I_7 := #VDReqPhoneAlarm[8],
                     I_8 := #VDReqPhoneAlarm[9],
                     I_9 := #VDReqPhoneAlarm[10],
                     I_10 := #VDReqPhoneAlarm[11],
                     I_11 := #VDReqPhoneAlarm[12],
                     I_12 := #VDReqPhoneAlarm[13],
                     I_13 := #VDReqPhoneAlarm[14],
                     I_14 := #VDReqPhoneAlarm[15],
                     I_15 := #VDReqPhoneAlarm[16],
                     I_16 := "FALSE",
                     I_17 := "FALSE",
                     I_18 := "FALSE",
                     I_19 := "FALSE",
                     I_20 := "FALSE",
                     I_21 := "FALSE",
                     I_22 := "FALSE",
                     I_23 := "FALSE",
                     I_24 := "FALSE",
                     I_25 := "FALSE",
                     I_26 := "FALSE",
                     I_27 := "FALSE",
                     I_28 := "FALSE",
                     I_29 := "FALSE",
                     I_30 := "FALSE",
                     I_31 := "FALSE",
                     O_DWord => #H_PhoneAlarmReqString.H_Anim.H_DWord);
   END_IF;
END_REGION

REGION Network 73: **** 4.6 - Machine status - Indication **** Animation Message
   IF "Blink_2,0s" THEN
       #H_PhoneAlarmReqString.H_Message[1] := #C_Message1;
       #H_PhoneAlarmReqString.H_Message[2] := #C_Message2;
       #H_PhoneAlarmReqString.H_Message[3] := #C_Message3;
       #H_PhoneAlarmReqString.H_Message[4] := #C_Message4;
       #H_PhoneAlarmReqString.H_Message[5] := #C_Message5;
       #H_PhoneAlarmReqString.H_Message[6] := #C_Message6;
       #H_PhoneAlarmReqString.H_Message[7] := #C_Message7;
       #H_PhoneAlarmReqString.H_Message[8] := #C_Message8;
       #H_PhoneAlarmReqString.H_Message[9] := #C_Message9;
       #H_PhoneAlarmReqString.H_Message[10] := #C_Message10;
       #H_PhoneAlarmReqString.H_Message[11] := #C_Message11;
       #H_PhoneAlarmReqString.H_Message[12] := #C_Message12;
       #H_PhoneAlarmReqString.H_Message[13] := #C_Message13;
       #H_PhoneAlarmReqString.H_Message[14] := #C_Message14;
       #H_PhoneAlarmReqString.H_Message[15] := #C_Message15;
       #H_PhoneAlarmReqString.H_Message[16] := #C_Message16;
   END_IF;
END_REGION

REGION Network 74: **** 4.6 - Machine status - Indication **** Animation Message Type
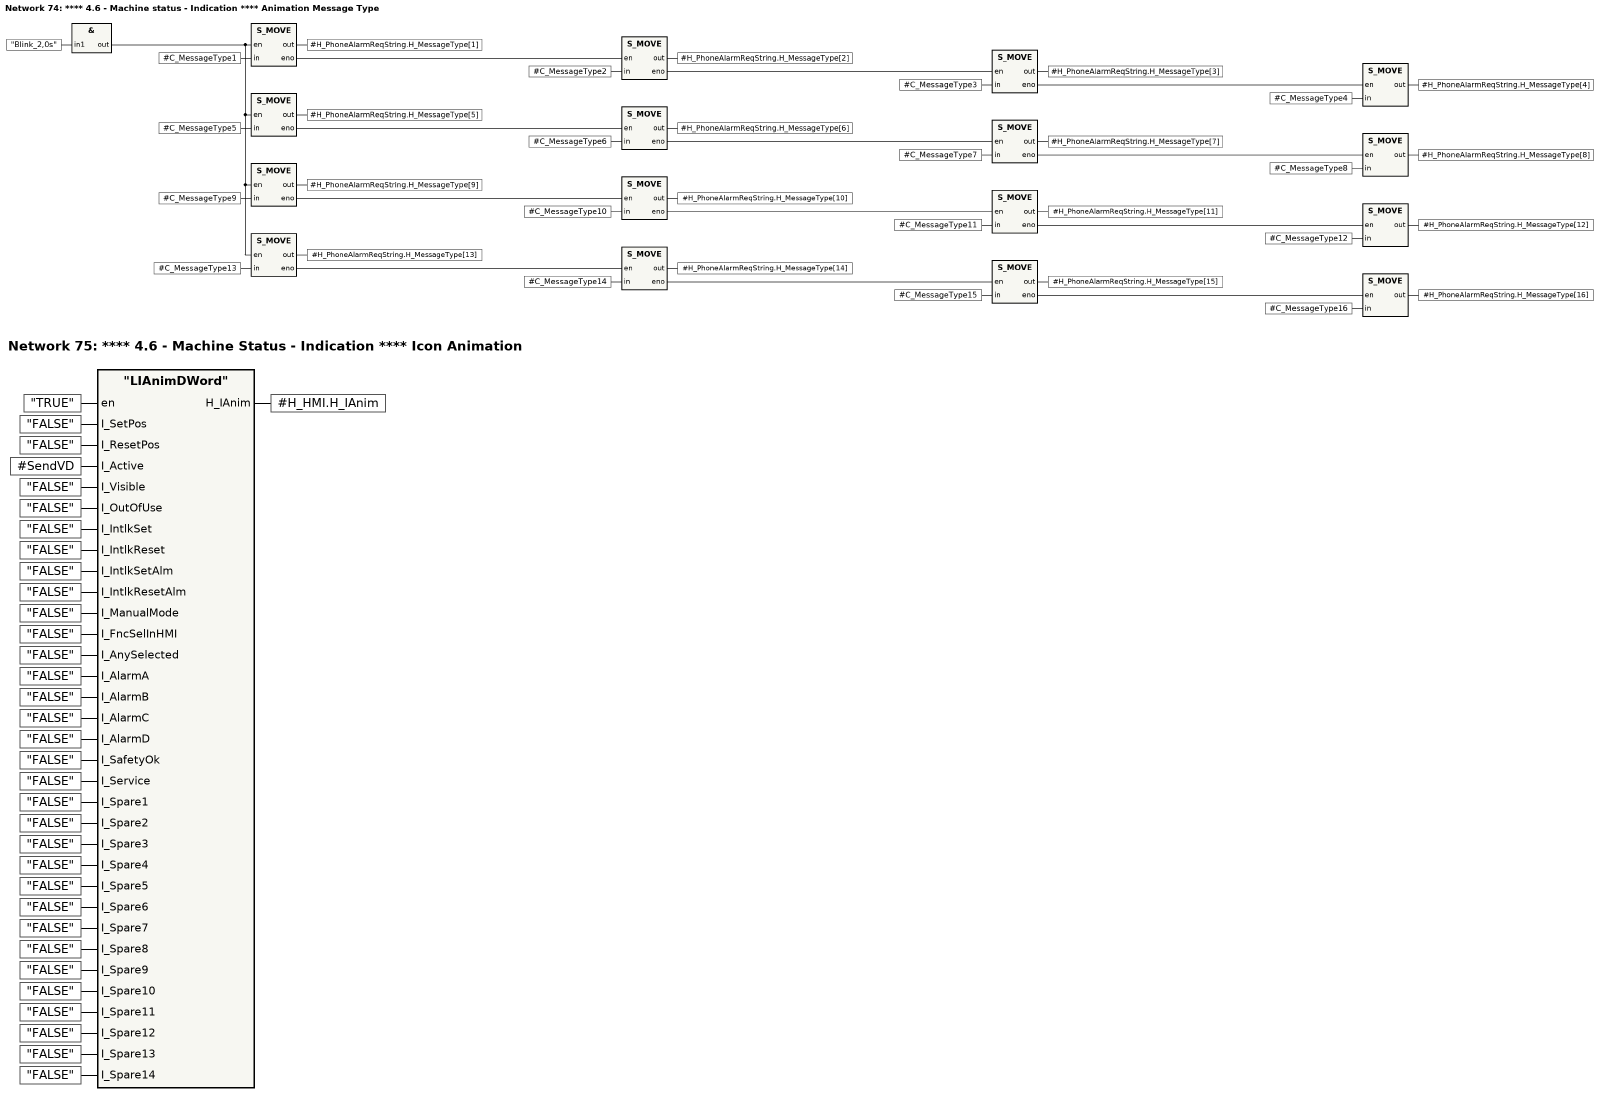
   IF "Blink_2,0s" THEN
       #H_PhoneAlarmReqString.H_MessageType[1] := #C_MessageType1;
       #H_PhoneAlarmReqString.H_MessageType[2] := #C_MessageType2;
       #H_PhoneAlarmReqString.H_MessageType[3] := #C_MessageType3;
       #H_PhoneAlarmReqString.H_MessageType[4] := #C_MessageType4;
       #H_PhoneAlarmReqString.H_MessageType[5] := #C_MessageType5;
       #H_PhoneAlarmReqString.H_MessageType[6] := #C_MessageType6;
       #H_PhoneAlarmReqString.H_MessageType[7] := #C_MessageType7;
       #H_PhoneAlarmReqString.H_MessageType[8] := #C_MessageType8;
       #H_PhoneAlarmReqString.H_MessageType[9] := #C_MessageType9;
       #H_PhoneAlarmReqString.H_MessageType[10] := #C_MessageType10;
       #H_PhoneAlarmReqString.H_MessageType[11] := #C_MessageType11;
       #H_PhoneAlarmReqString.H_MessageType[12] := #C_MessageType12;
       #H_PhoneAlarmReqString.H_MessageType[13] := #C_MessageType13;
       #H_PhoneAlarmReqString.H_MessageType[14] := #C_MessageType14;
       #H_PhoneAlarmReqString.H_MessageType[15] := #C_MessageType15;
       #H_PhoneAlarmReqString.H_MessageType[16] := #C_MessageType16;
   END_IF;
END_REGION

REGION Network 75: **** 4.6 - Machine Status - Indication **** Icon Animation
   // Icon Animation
   IF "TRUE" THEN
       "LIAnimDWord"(I_SetPos := "FALSE",
                     I_ResetPos := "FALSE",
                     I_Active := #SendVD,
                     I_Visible := "FALSE",
                     I_OutOfUse := "FALSE",
                     I_IntlkSet := "FALSE",
                     I_IntlkReset := "FALSE",
                     I_IntlkSetAlm := "FALSE",
                     I_IntlkResetAlm := "FALSE",
                     I_ManualMode := "FALSE",
                     I_FncSelInHMI := "FALSE",
                     I_AnySelected := "FALSE",
                     I_AlarmA := "FALSE",
                     I_AlarmB := "FALSE",
                     I_AlarmC := "FALSE",
                     I_AlarmD := "FALSE",
                     I_SafetyOk := "FALSE",
                     I_Service := "FALSE",
                     I_Spare1 := "FALSE",
                     I_Spare2 := "FALSE",
                     I_Spare3 := "FALSE",
                     I_Spare4 := "FALSE",
                     I_Spare5 := "FALSE",
                     I_Spare6 := "FALSE",
                     I_Spare7 := "FALSE",
                     I_Spare8 := "FALSE",
                     I_Spare9 := "FALSE",
                     I_Spare10 := "FALSE",
                     I_Spare11 := "FALSE",
                     I_Spare12 := "FALSE",
                     I_Spare13 := "FALSE",
                     I_Spare14 := "FALSE",
                     H_IAnim => #H_HMI.H_IAnim);
   END_IF;
END_REGION

REGION Network 76: **** 8 - Outputs **** Data / **** 8 - Outputs **** Prepare Data
   // Data / Prepare Data
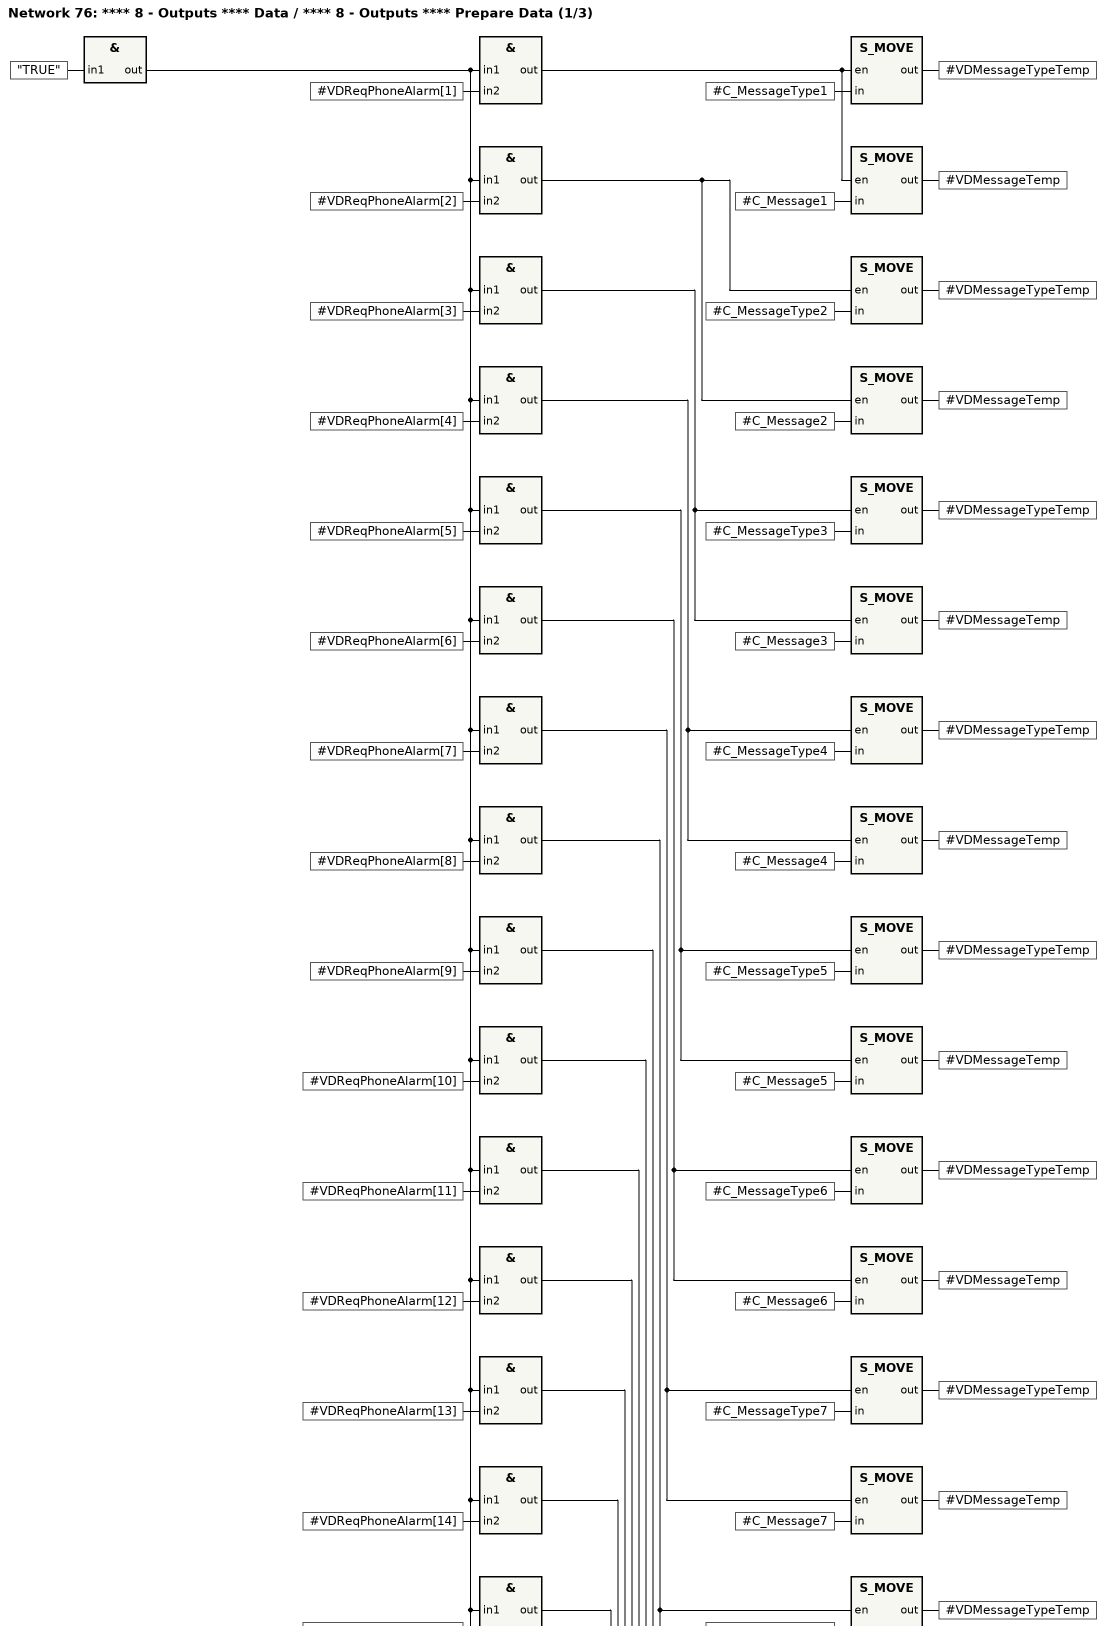
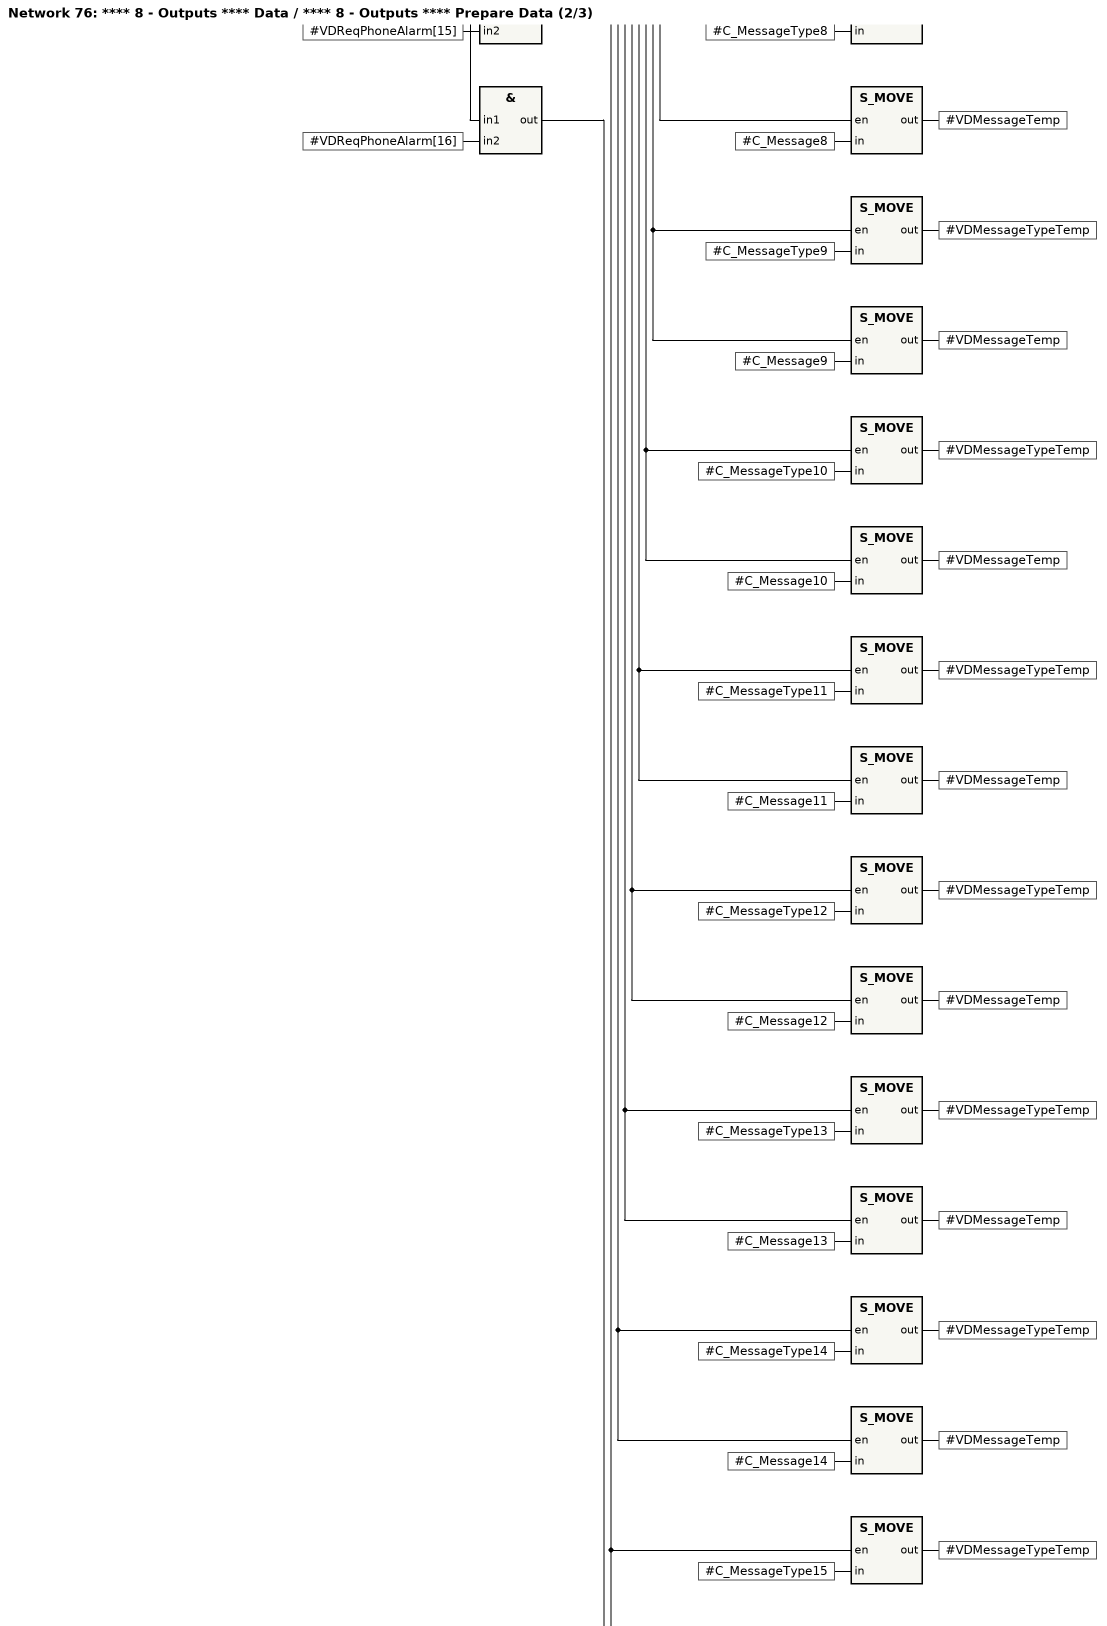
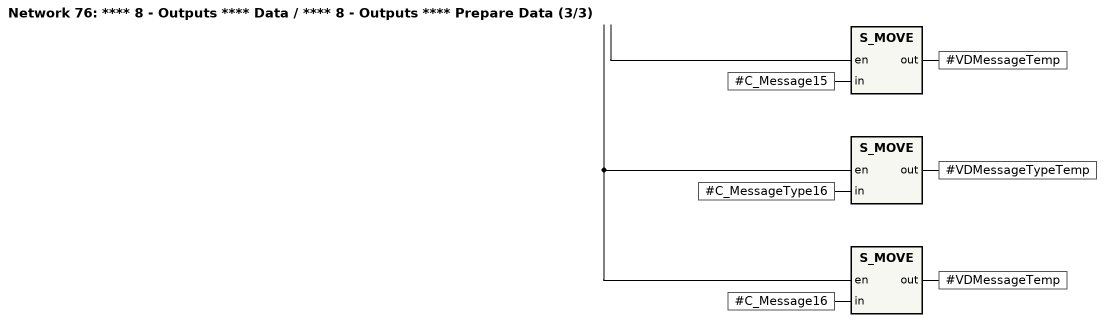
   IF "TRUE" AND #VDReqPhoneAlarm[1] THEN
       #VDMessageTypeTemp := #C_MessageType1;
       #VDMessageTemp := #C_Message1;
   END_IF;
   IF "TRUE" AND #VDReqPhoneAlarm[2] THEN
       #VDMessageTypeTemp := #C_MessageType2;
       #VDMessageTemp := #C_Message2;
   END_IF;
   IF "TRUE" AND #VDReqPhoneAlarm[3] THEN
       #VDMessageTypeTemp := #C_MessageType3;
       #VDMessageTemp := #C_Message3;
   END_IF;
   IF "TRUE" AND #VDReqPhoneAlarm[4] THEN
       #VDMessageTypeTemp := #C_MessageType4;
       #VDMessageTemp := #C_Message4;
   END_IF;
   IF "TRUE" AND #VDReqPhoneAlarm[5] THEN
       #VDMessageTypeTemp := #C_MessageType5;
       #VDMessageTemp := #C_Message5;
   END_IF;
   IF "TRUE" AND #VDReqPhoneAlarm[6] THEN
       #VDMessageTypeTemp := #C_MessageType6;
       #VDMessageTemp := #C_Message6;
   END_IF;
   IF "TRUE" AND #VDReqPhoneAlarm[7] THEN
       #VDMessageTypeTemp := #C_MessageType7;
       #VDMessageTemp := #C_Message7;
   END_IF;
   IF "TRUE" AND #VDReqPhoneAlarm[8] THEN
       #VDMessageTypeTemp := #C_MessageType8;
       #VDMessageTemp := #C_Message8;
   END_IF;
   IF "TRUE" AND #VDReqPhoneAlarm[9] THEN
       #VDMessageTypeTemp := #C_MessageType9;
       #VDMessageTemp := #C_Message9;
   END_IF;
   IF "TRUE" AND #VDReqPhoneAlarm[10] THEN
       #VDMessageTypeTemp := #C_MessageType10;
       #VDMessageTemp := #C_Message10;
   END_IF;
   IF "TRUE" AND #VDReqPhoneAlarm[11] THEN
       #VDMessageTypeTemp := #C_MessageType11;
       #VDMessageTemp := #C_Message11;
   END_IF;
   IF "TRUE" AND #VDReqPhoneAlarm[12] THEN
       #VDMessageTypeTemp := #C_MessageType12;
       #VDMessageTemp := #C_Message12;
   END_IF;
   IF "TRUE" AND #VDReqPhoneAlarm[13] THEN
       #VDMessageTypeTemp := #C_MessageType13;
       #VDMessageTemp := #C_Message13;
   END_IF;
   IF "TRUE" AND #VDReqPhoneAlarm[14] THEN
       #VDMessageTypeTemp := #C_MessageType14;
       #VDMessageTemp := #C_Message14;
   END_IF;
   IF "TRUE" AND #VDReqPhoneAlarm[15] THEN
       #VDMessageTypeTemp := #C_MessageType15;
       #VDMessageTemp := #C_Message15;
   END_IF;
   IF "TRUE" AND #VDReqPhoneAlarm[16] THEN
       #VDMessageTypeTemp := #C_MessageType16;
       #VDMessageTemp := #C_Message16;
   END_IF;
END_REGION

REGION Network 77: **** 8 - Outputs **** Prepare MessageType and Message
   // Prepare Message
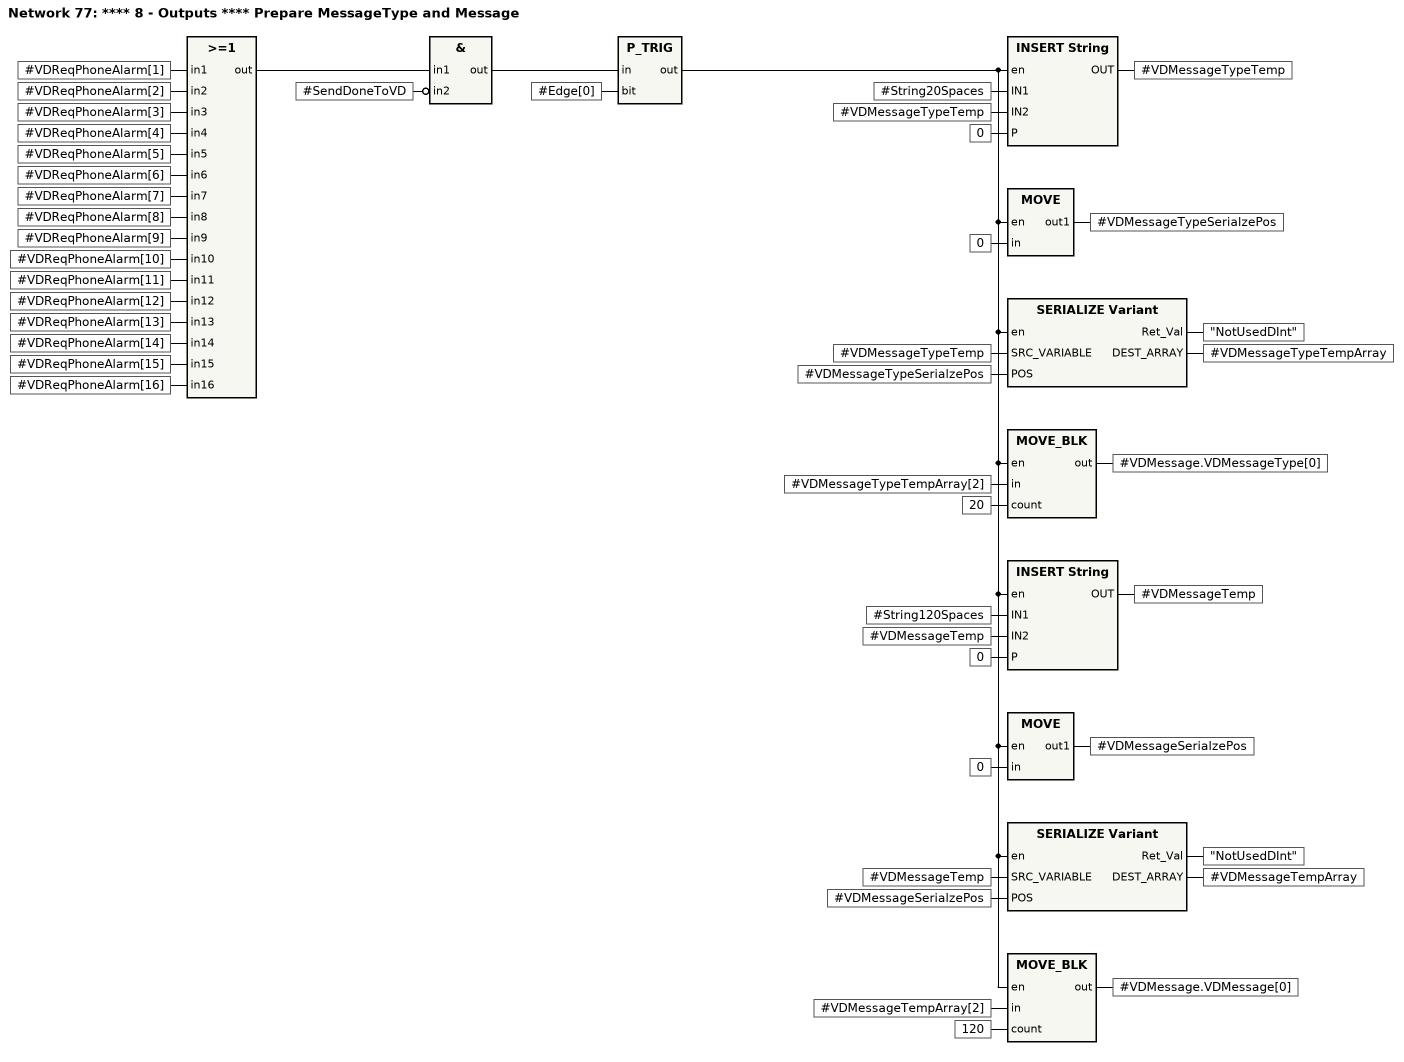
   #_w1 := (#VDReqPhoneAlarm[1] OR #VDReqPhoneAlarm[2] OR #VDReqPhoneAlarm[3] OR #VDReqPhoneAlarm[4] OR #VDReqPhoneAlarm[5] OR #VDReqPhoneAlarm[6] OR #VDReqPhoneAlarm[7] OR #VDReqPhoneAlarm[8] OR #VDReqPhoneAlarm[9] OR #VDReqPhoneAlarm[10] OR #VDReqPhoneAlarm[11] OR #VDReqPhoneAlarm[12] OR #VDReqPhoneAlarm[13] OR #VDReqPhoneAlarm[14] OR #VDReqPhoneAlarm[15] OR #VDReqPhoneAlarm[16]) AND NOT #SendDoneToVD;
   #_w2 := #_w1 AND NOT #Edge[0];   // rising edge
   #Edge[0] := #_w1;
   IF #_w2 THEN
       INSERT(IN1 := #String20Spaces, IN2 := #VDMessageTypeTemp, P := 0, OUT => #VDMessageTypeTemp);
       #VDMessageTypeSerialzePos := 0;
       "NotUsedDInt" := Serialize(SRC_VARIABLE := #VDMessageTypeTemp,
                               POS := #VDMessageTypeSerialzePos,
                               DEST_ARRAY => #VDMessageTypeTempArray);
       MOVE_BLK(IN := #VDMessageTypeTempArray[2], COUNT := 20, OUT => #VDMessage.VDMessageType[0]);
       INSERT(IN1 := #String120Spaces, IN2 := #VDMessageTemp, P := 0, OUT => #VDMessageTemp);
       #VDMessageSerialzePos := 0;
       "NotUsedDInt" := Serialize(SRC_VARIABLE := #VDMessageTemp,
                               POS := #VDMessageSerialzePos,
                               DEST_ARRAY => #VDMessageTempArray);
       MOVE_BLK(IN := #VDMessageTempArray[2], COUNT := 120, OUT => #VDMessage.VDMessage[0]);
   END_IF;
END_REGION

REGION Network 78: **** 8 - Outputs **** Send To VD
   // Send To VD
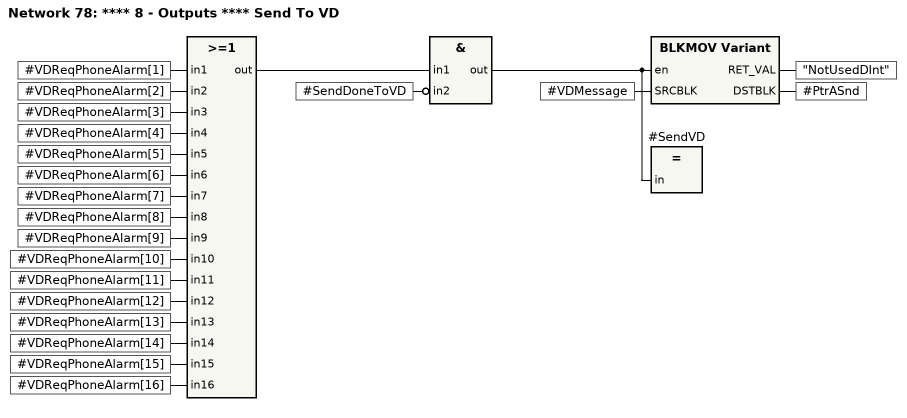
   #_w1 := (#VDReqPhoneAlarm[1] OR #VDReqPhoneAlarm[2] OR #VDReqPhoneAlarm[3] OR #VDReqPhoneAlarm[4] OR #VDReqPhoneAlarm[5] OR #VDReqPhoneAlarm[6] OR #VDReqPhoneAlarm[7] OR #VDReqPhoneAlarm[8] OR #VDReqPhoneAlarm[9] OR #VDReqPhoneAlarm[10] OR #VDReqPhoneAlarm[11] OR #VDReqPhoneAlarm[12] OR #VDReqPhoneAlarm[13] OR #VDReqPhoneAlarm[14] OR #VDReqPhoneAlarm[15] OR #VDReqPhoneAlarm[16]) AND NOT #SendDoneToVD;
   IF #_w1 THEN "NotUsedDInt" := BLKMOV(SRCBLK := #VDMessage, DSTBLK => #PtrASnd); END_IF;
   #SendVD := #_w1;
END_REGION
END_FUNCTION_BLOCK
